(* ---------------------- Limitation of the command signal between +/- SpeedLimit ----------------------------*)
IF fL_CommandSignal > (fI_SpeedLimit) THEN
  fL_CommandSignal :=  fI_SpeedLimit;
ELSIF fL_CommandSignal < (-fI_SpeedLimit) THEN
  fL_CommandSignal := -fI_SpeedLimit;
END_IF;

IF bI_MoveEnable THEN
  IF fI_Microstepping <> 0 THEN
    iO_TargetVelocity := FC_REAL_TO_INT((fI_LimitSpeedFullStep / (fI_LimitSpeedFullStep / fI_Microstepping / 60 * fI_Axis_Scaling) * fL_CommandSignal * fL_PercentageRampUP)); 
    //iO_TargetVelocity := FC_REAL_TO_INT((fI_SpeedScaling / fI_Axis_Scaling * fL_CommandSignal * fL_PercentageRampUP));      (* Send the Target velocity command to module *)
  END_IF;
ELSE
  IF fI_Microstepping <> 0 THEN
    iO_TargetVelocity := FC_REAL_TO_INT((fI_LimitSpeedFullStep / (fI_LimitSpeedFullStep / fI_Microstepping / 60 * fI_Axis_Scaling) * fL_CommandSignal * (1-fL_PercentageRampDN))); 
    //iO_TargetVelocity := FC_REAL_TO_INT((fI_SpeedScaling / fI_Axis_Scaling * fL_CommandSignal * (1-fL_PercentageRampDN)));  (* Send the Target velocity command to module *)
  END_IF;
END_IF;

IF NOT bI_EStop THEN
  iO_TargetVelocity := 0;
END_IF;


(* ---------------------- Encoder Offset Calibration ----------------- *)

IF bI_SetPosition AND NOT bL_memSetPosition AND NOT bI_MoveEnable THEN
  IF fI_Axis_Scaling <> 0 THEN
    fL_OffsetEncoder := FC_REAL_TO_DINT((fI_SetPositionValue * fI_EncoderScaling / fI_Axis_Scaling - DINT_TO_REAL(lI_EncoderValue)));
  END_IF;

  fL_memTargetPosition := fO_ActualPosition;
END_IF;

(* ---------------------- Memory ----------------- *)
bL_memSetPosition := bI_SetPosition;
bL_memMoveEnable  := bI_MoveEnable;
bL_FirstRun       := FALSE;

(********************************* END OF FB *****************************************************)

METHOD PRIVATE Input
VAR_INPUT
END_VAR
(*EL7041 Standard: 20 Singleturn bits and 12 Multiturn bits*)
IF (fI_EncoderScaling <> 0) THEN
	fO_ActualPosition := (DINT_TO_REAL(lI_EncoderValue) + DINT_TO_REAL(fL_OffsetEncoder)) * fI_Axis_Scaling / fI_EncoderScaling;
END_IF;

(*Movement done?*)
IF bI_MoveEnable THEN
	IF ABS(fL_memTargetPosition - fO_ActualPosition) < fI_Tolerance * 0.2 THEN
		bO_MoveOK := TRUE;
	ELSE
		bO_MoveOK := FALSE;
	END_IF;
ELSE
	IF ABS(fL_memTargetPosition - fO_ActualPosition) < fI_Tolerance THEN
		bO_MoveOK := TRUE;
	ELSE
		bO_MoveOK := FALSE;
	END_IF;
END_IF;
END_METHOD

END_FUNCTION_BLOCK

// ---- POUs/Machine/CleaningStation/FB_EL7201_001_AXIS_CTRL.TcPOU
FUNCTION_BLOCK FB_EL7201_001_AXIS_CTRL
(*************************************************************************************************)
(*  FILENAME:    FB_EL7201_001_AXIS_CTRL.EXP                                                     *)
(*  PROJECT:     CALMAR PUPLC                                                                    *)
(*  COPYRIGHT:   All rights reserved (c) Wifag//Polytype, Fribourg/Switzerland (2016)            *)
(*  ENVIRONMENT: TwinCAT PLC                                                                     *)
(*  VERSION:     <version>                                                                       *)
(*************************************************************************************************)
(*  DESCRIPTION:                                                                   <description> *)
(*     This function transfers the movement commands to the motor.                               *)
(*     It also controls the states of the EL7201 for the Cleaning Unit.                          *)
(*                                                                                </description> *)
(*************************************************************************************************)

{library public}
VAR_INPUT
  fI_TargetPosition              : REAL;                         (*Target position*)
  fI_Tolerance                   : REAL := 0.00002;              (*Position tolerance*)
  fI_SpeedLimit                  : REAL;                         (*Speed limit*)
  bI_MoveEnable                  : BOOL;                         (*Enable movement*)
  bI_RegActive                   : BOOL;                         (*Regulation active*)
  bI_FaultReset                  : BOOL;                         (*Fault reset*)
  bI_EStop                       : BOOL;                         (*Emergency stop*)
  bI_SetPosition                 : BOOL;                         (*Set position*)

  wI_StatusWord                  : UINT;                         (*Status word: 6041:0*)
  lI_EncoderValue                : UDINT;                        (*Encoder value*)
  fI_PosControllerGain           : REAL := 1.0;                  (*Position controller gain*)
  fI_EncoderScaling              : REAL := 1048576;              (*Encoder scaling [counts/rev]*)
  fI_Axis_Scaling                : REAL := 0.0002;               (*Axis scaling [m/rev]*)
  fI_SetPositionValue            : REAL := 0.0;                  (*Set position value [m]*)
  fI_SpeedScaling                : REAL := 268435;               (*Speed scaling [counts/rev]*)

  pI_OffsetEncoder               : POINTER TO DINT;              (*Offset to remanent value in encoder*)
END_VAR

VAR_OUTPUT
  wO_ControlWord                 : UINT;                         (*Control word:  6040:0*)
  iO_TargetVelocity              : DINT;                         (*Target velocity:  60FF:0*)
  fO_ActualPosition              : REAL;                         (*Actual position [m]*)
  bO_MoveOk                      : BOOL;                         (*Movement ok*)
  eO_EL7201Status                : EN_EL7201_STATE;              (*EL7201 Status*)
  bO_AxisNotInit                 : BOOL;                         (*Axis not initialized*)
END_VAR

{library private}
VAR
  fL_Delta_P                     : REAL;                         (*Delta position*)
  fL_CommandSignal               : REAL;                         (*Command signal*)

  tL_TimerRampUP                 : TON;                          (*Timer ramp up*)
  fL_PercentageRampUP            : REAL;                         (*Percentage ramp up*)
  tL_TimerRampDN                 : TON;                          (*Timer ramp down*)
  fL_PercentageRampDN            : REAL;                         (*Percentage ramp down*)

  wL_MaskedStatusWord            : WORD;                         (*Masked status word*)
  bL_memMoveEnable               : BOOL;                         (*Memory enable movement*)
  bL_memSetPosition              : BOOL;                         (*Memory set position*)
  fL_memTargetPosition           : REAL := 0.0;                  (*Memory target position*)
  bL_StopRamp                    : BOOL;                         (*Stop ramp*)
  bL_FirstRun                    : BOOL := TRUE;                 (*First run*)

  fL_Divider                     : REAL;                         (*Divider for percent calculation*)
END_VAR

Input();

tL_TimerRampUP.PT :=T#100ms;
tL_TimerRampUP();

tL_TimerRampDN.PT :=T#100ms;
tL_TimerRampDN();

IF bI_MoveEnable=FALSE AND bL_memMoveEnable THEN
	bL_StopRamp := TRUE;
END_IF;

IF bI_MoveEnable AND NOT bL_memMoveEnable THEN
	fL_memTargetPosition := fI_TargetPosition;
	bO_MoveOK := FALSE;
ELSIF bL_FirstRun THEN
	fL_memTargetPosition := fO_ActualPosition;
END_IF;


IF tL_TimerRampDN.Q THEN
	bL_StopRamp:=FALSE;
END_IF;

tL_TimerRampDN.IN := bL_StopRamp;

fL_Divider := TIME_TO_REAL(tL_TimerRampDN.PT);
IF fL_Divider <> 0 THEN
	fL_PercentageRampDN := TIME_TO_REAL(tL_TimerRampDN.ET)/fL_Divider;
END_IF;

tL_TimerRampUP.IN := bI_MoveEnable AND bI_RegActive;

fL_Divider := TIME_TO_REAL(tL_TimerRampUP.PT);
IF fL_Divider <> 0 THEN
	fL_PercentageRampUP := TIME_TO_REAL(tL_TimerRampUP.ET)/fL_Divider;
END_IF;

(* ---------------------- Calculation of the Error Signal between the Target and the Actual Position -----------------*)
fL_Delta_P := fI_TargetPosition - fO_ActualPosition;

(* --------------------------------- Calculation of the Command Signal for the Target Velocity  ---------------------------*)
fL_CommandSignal := fL_Delta_P * fI_PosControllerGain;

(* ----------------------------- Limitation of the Command Signal between +/- SpeedLimit --------------------------------*)
IF fL_CommandSignal > (fI_SpeedLimit) THEN
	fL_CommandSignal:= fI_SpeedLimit;
ELSIF fL_CommandSignal < (-fI_SpeedLimit) THEN
	fL_CommandSignal:=-fI_SpeedLimit;
END_IF;

IF bI_MoveEnable THEN
	IF fI_Axis_Scaling <> 0 THEN
		iO_TargetVelocity:= FC_REAL_TO_DINT((fI_SpeedScaling / fI_Axis_Scaling * fL_CommandSignal * fL_PercentageRampUP));			(* Send the Target velocity command to module *)
	END_IF;
ELSE
	IF fI_Axis_Scaling <> 0 THEN
		iO_TargetVelocity:= FC_REAL_TO_DINT((fI_SpeedScaling / fI_Axis_Scaling * fL_CommandSignal * (1-fL_PercentageRampDN)));	(* Send the Target velocity command to module *)
	END_IF;
END_IF;
(* ---------------------- MDP StateMachine ----------------- *)

wL_MaskedStatusWord := UINT_TO_WORD(wI_StatusWord) AND 16#006F;

IF bI_EStop=FALSE THEN
	iO_TargetVelocity:=0;
	eO_EL7201Status := eEstopped;
	wO_ControlWord := 16#0000;
	wO_ControlWord := 16#0002;
ELSE

	CASE wL_MaskedStatusWord OF
			16#0000, 16#0020:								(* ------------------ State : Not Ready to Switch On : x0xx0000 ---------------------- *)
				eO_EL7201Status := eNotReadyToSwitchON ;

			16#0040, 16#0060:								(* ------------------ State : Switch ON Disable : x1xx0000 ---------------------- *)
				eO_EL7201Status := eSwitchONDisabled ;
				wO_ControlWord := 16#0006;

			16#0021:										(* ------------------ State : Ready To Switch ON : x01x0001---------------------- *)
				eO_EL7201Status := eReadyToSwitchON ;
				IF bI_RegActive=TRUE THEN
					wO_ControlWord := 16#0007;
				ELSE
					wO_ControlWord := 16#0006;
				END_IF;

			16#0023:										(* ---------------- State : Switched ON : x01x0011------------------ *)
				eO_EL7201Status := eSwitchedON ;
				IF bI_MoveEnable=TRUE THEN
					wO_ControlWord := 16#000F;
				END_IF;

				IF bI_RegActive=FALSE THEN
					wO_ControlWord := 16#0006;
				END_IF;

			16#0027:										(* -------------- State : Enabled : x01x0111------------------ *)
				eO_EL7201Status := eEnabled;
				IF (bI_MoveEnable=FALSE AND tL_TimerRampDN.Q) THEN
					wO_ControlWord := 16#0007;
				END_IF;

			16#000F, 16#002F:								(* -------------- State : Fault Reaction Active : x0xx1111----------------- *)
				eO_EL7201Status := eFaultReactionActive ;

			16#0008, 16#0028, 16#0068:								(* --------------- State :  Fault : x0xx1000 ------------------- *)
				eO_EL7201Status := eFault;
				IF bI_FaultReset THEN
					wO_ControlWord := 16#0080;
				ELSE
					wO_ControlWord := 16#0000;
				END_IF;
	END_CASE;
END_IF;

(* ---------------------- Encoder Offset Calibration ----------------- *)

IF bI_SetPosition AND NOT bL_memSetPosition AND NOT bI_MoveEnable THEN
	IF fI_Axis_Scaling <> 0 THEN
		pI_OffsetEncoder^:= FC_REAL_TO_DINT((fI_SetPositionValue * fI_EncoderScaling / fI_Axis_Scaling - UDINT_TO_REAL(lI_EncoderValue)));
	END_IF;

	fL_memTargetPosition := fO_ActualPosition;
END_IF;

IF pI_OffsetEncoder^ = 0 OR pI_OffsetEncoder = 0 THEN
	bO_AxisNotInit := TRUE;
ELSE
	bO_AxisNotInit := FALSE;
END_IF;

(* ---------------------- Memory ----------------- *)
bL_memSetPosition := bI_SetPosition;
bL_memMoveEnable  := bI_MoveEnable;
bL_FirstRun       := FALSE;

(********************************* END OF FB *****************************************************)

ACTION Input:
(*EL7201 Standard: 20 Singleturn bits and 12 Multiturn bits*)
IF fI_EncoderScaling <> 0 AND pI_OffsetEncoder <> 0 THEN
	fO_ActualPosition:=(UDINT_TO_REAL(lI_EncoderValue) + DINT_TO_REAL(pI_OffsetEncoder^)) * fI_Axis_Scaling / fI_EncoderScaling;
END_IF;

(*Movement done?*)
IF ABS(fL_memTargetPosition - fO_ActualPosition) < fI_Tolerance THEN
	bO_MoveOK := TRUE;
ELSE
	bO_MoveOK := FALSE;
END_IF;

(********************************* END OF ACTION *************************************************)
END_ACTION

END_FUNCTION_BLOCK

// ---- POUs/Machine/CleaningStation/FB_EL7201_AXIS_CTRL.TcPOU
FUNCTION_BLOCK FB_EL7201_AXIS_CTRL
(*************************************************************************************************)
(*  FILENAME:    FB_EL7201_AXIS_CTRL.EXP                                                         *)
(*  PROJECT:     CALMAR PUPLC                                                                    *)
(*  COPYRIGHT:   All rights reserved (c) Wifag//Polytype, Fribourg/Switzerland (2016)            *)
(*  ENVIRONMENT: TwinCAT PLC                                                                     *)
(*  VERSION:     <version>                                                                       *)
(*************************************************************************************************)
(*  DESCRIPTION:                                                                   <description> *)
(*     This function transfers the movement commands to the motor.                               *)
(*     It also controls the states of the EL7201 for the Cleaning Unit.                          *)
(*                                                                                </description> *)
(*************************************************************************************************)

{library public}
VAR_INPUT
  fI_TargetPosition              : REAL;                         (*Target position*)
  fI_Tolerance                   : REAL := 0.0001;               (*Position tolerance*)
  fI_SpeedLimit                  : REAL;                         (*Speed limit*)
  bI_MoveEnable                  : BOOL;                         (*Enable movement*)
  bI_RegActive                   : BOOL;                         (*Regulation active*)
  bI_FaultReset                  : BOOL;                         (*Fault reset*)
  bI_MsgReset                    : BOOL;                         (*Message reset*)
  bI_EStop                       : BOOL;                         (*Emergency stop*)
  bI_SetPosition                 : BOOL;                         (*Set position*)

  wI_StatusWord                  : UINT;                         (*Status word: 6041:0*)
  lI_EncoderValue                : DINT;                         (*Encoder value*)
  fI_PosControllerGain           : REAL := 1.0;                  (*Position controller gain*)
  fI_EncoderScaling              : REAL := 1048576;              (*Encoder scaling [counts/rev]*)
  fI_Axis_Scaling                : REAL := 0.0002;               (*Axis scaling [m/rev]*)
  fI_SetPositionValue            : REAL := 0.0;                  (*Set position value [m]*)
  fI_SpeedScaling                : REAL := 268435;               (*Speed scaling [counts/rev]*)

  pI_OffsetEncoder               : POINTER TO DINT;              (*Offset to remanent value in encoder*)

  fI_TolDriveTimeFactor          : REAL := 2.0;                  (*Factor for tolerated drive time*)
END_VAR

VAR_OUTPUT
  wO_ControlWord                 : UINT;                         (*Control word:  6040:0*)
  iO_TargetVelocity              : DINT;                         (*Target velocity:  60FF:0*)
  fO_ActualPosition              : REAL;                         (*Actual position [m]*)
  bO_MoveOk                      : BOOL;                         (*Movement ok*)
  eO_EL7201Status                : EN_EL7201_STATE;              (*EL7201 status*)
  bO_WarnDriveTime               : BOOL;                         (*Error drive time too long*)
END_VAR

{library private}
VAR
  fL_Delta_P                     : REAL;                         (*Delta position*)
  fL_CommandSignal               : REAL;                         (*Command signal*)

  tL_TimerRampUP                 : TON;                          (*Timer ramp up*)
  fL_PercentageRampUP            : REAL;                         (*Percentage ramp up*)
  tL_TimerRampDN                 : TON;                          (*Timer ramp down*)
  fL_PercentageRampDN            : REAL;                         (*Percentage ramp down*)

  wL_MaskedStatusWord            : WORD;                         (*Masked status word*)
  bL_memMoveEnable               : BOOL;                         (*Memory enable movement*)
  bL_memSetPosition              : BOOL;                         (*Memory set position*)
  fL_memTargetPosition           : REAL := 0.0;                  (*Memory target position*)
  bL_StopRamp                    : BOOL;                         (*Stop ramp*)
  bL_FirstRun                    : BOOL := TRUE;                 (*First run*)

  fL_Divider                     : REAL;                         (*Divider for percent calculation*)
  
  fb_RTrigEnable                 : R_TRIG;                       (*RTrig for motor enable*)
  fL_CalcDriveTime               : REAL;                         (*Calculated drive time [s]*)
  fL_RampDriveTime               : REAL := 10;                   (*Ramp time [s]*)
  tL_DriveTime                   : TON;                          (*Timer drive time*)
  iL_SpeedNotSetCounter          : UINT;                         (*Debug: speed limit for calculation not set*)
END_VAR

Input();

tL_TimerRampUP.PT :=T#300ms;
tL_TimerRampUP();

tL_TimerRampDN.PT :=T#300ms;
tL_TimerRampDN();

IF bI_MoveEnable=FALSE AND bL_memMoveEnable=TRUE THEN
	bL_StopRamp := TRUE;
END_IF;

IF bI_MoveEnable=TRUE AND bL_memMoveEnable=FALSE THEN
	fL_memTargetPosition := fI_TargetPosition;
	bO_MoveOK := FALSE;
ELSIF bL_FirstRun THEN
	fL_memTargetPosition := fO_ActualPosition;
END_IF;


IF tL_TimerRampDN.Q THEN
	bL_StopRamp:=FALSE;
END_IF;

tL_TimerRampDN.IN := bL_StopRamp;

fL_Divider := TIME_TO_REAL(tL_TimerRampDN.PT);
IF fL_Divider <> 0 THEN
	fL_PercentageRampDN := TIME_TO_REAL(tL_TimerRampDN.ET)/fL_Divider;
END_IF;

tL_TimerRampUP.IN := bI_MoveEnable AND bI_RegActive;

fL_Divider := TIME_TO_REAL(tL_TimerRampUP.PT);
IF fL_Divider <> 0 THEN
	fL_PercentageRampUP := TIME_TO_REAL(tL_TimerRampUP.ET)/fL_Divider;
END_IF;

(* ---------------------- Calculation of the Error Signal between the Target and the Actual Position -----------------*)
fL_Delta_P := fI_TargetPosition - fO_ActualPosition;

(* --------------------------------- Calculation of the Command Signal for the Target Velocity  ---------------------------*)
fL_CommandSignal := fL_Delta_P * fI_PosControllerGain;

(* ----------------------------- Limitation of the Command Signal between +/- SpeedLimit --------------------------------*)
IF fL_CommandSignal > (fI_SpeedLimit) THEN
	fL_CommandSignal:= fI_SpeedLimit;
ELSIF fL_CommandSignal < (-fI_SpeedLimit) THEN
	fL_CommandSignal:=-fI_SpeedLimit;
END_IF;

IF bI_MoveEnable THEN
	IF fI_Axis_Scaling <> 0 THEN
		iO_TargetVelocity:= FC_REAL_TO_DINT((fI_SpeedScaling / fI_Axis_Scaling * fL_CommandSignal * fL_PercentageRampUP));			(* Send the Target velocity command to module *)
	END_IF;
ELSE
	IF fI_Axis_Scaling <> 0 THEN
		iO_TargetVelocity:= FC_REAL_TO_DINT((fI_SpeedScaling / fI_Axis_Scaling * fL_CommandSignal * (1-fL_PercentageRampDN)));	(* Send the Target velocity command to module *)
	END_IF;
END_IF;
(* ---------------------- MDP StateMachine ----------------- *)

wL_MaskedStatusWord := UINT_TO_WORD(wI_StatusWord) AND 16#006F;

IF bI_EStop=FALSE THEN
	iO_TargetVelocity:=0;
	eO_EL7201Status := eEstopped;
	wO_ControlWord := 16#0000;
	wO_ControlWord := 16#0002;
ELSE

	CASE wL_MaskedStatusWord OF
			16#0000, 16#0020:								(* ------------------ State : Not Ready to Switch On : x0xx0000 ---------------------- *)
				eO_EL7201Status := eNotReadyToSwitchON ;

			16#0040, 16#0060:								(* ------------------ State : Switch ON Disable : x1xx0000 ---------------------- *)
				eO_EL7201Status := eSwitchONDisabled ;
				wO_ControlWord := 16#0006;

			16#0021:										(* ------------------ State : Ready To Switch ON : x01x0001---------------------- *)
				eO_EL7201Status := eReadyToSwitchON ;
				IF bI_RegActive=TRUE THEN
					wO_ControlWord := 16#0007;
				END_IF;

			16#0023:										(* ---------------- State : Switched ON : x01x0011------------------ *)
				eO_EL7201Status := eSwitchedON ;
				IF bI_MoveEnable=TRUE THEN
					wO_ControlWord := 16#000F;
				END_IF;

				IF bI_RegActive=FALSE THEN
					wO_ControlWord := 16#0006;
				END_IF;

			16#0027:										(* -------------- State : Enabled : x01x0111------------------ *)
				eO_EL7201Status := eEnabled;
				IF (bI_MoveEnable=FALSE AND tL_TimerRampDN.Q) THEN
					wO_ControlWord := 16#0007;
				END_IF;

			16#000F, 16#002F:								(* -------------- State : Fault Reaction Active : x0xx1111----------------- *)
				eO_EL7201Status := eFaultReactionActive ;

			16#0008, 16#0028, 16#0068:								(* --------------- State :  Fault : x0xx1000 ------------------- *)
				eO_EL7201Status := eFault;
				IF bI_FaultReset THEN
					wO_ControlWord := 16#0080;
				ELSE
					wO_ControlWord := 16#0000;
				END_IF;
	END_CASE;
END_IF;

(* ---------------------- Encoder Offset Calibration ----------------- *)

IF bI_SetPosition AND NOT bL_memSetPosition AND NOT bI_MoveEnable THEN
	IF fI_Axis_Scaling <> 0 THEN
		pI_OffsetEncoder^ := FC_REAL_TO_DINT((fI_SetPositionValue * fI_EncoderScaling / fI_Axis_Scaling - DINT_TO_REAL(lI_EncoderValue)));
	END_IF;

	fL_memTargetPosition := fO_ActualPosition;
END_IF;

(* ---------------------- Memory ----------------- *)
bL_memSetPosition := bI_SetPosition;
bL_memMoveEnable  := bI_MoveEnable;
bL_FirstRun       := FALSE;

(* ---------------------- Check motor for stiffness or blocking ----------------- *)
fb_RTrigEnable(CLK := bI_MoveEnable);
IF fb_RTrigEnable.Q THEN
  IF (fI_SpeedLimit <> 0) THEN
    fL_CalcDriveTime := ABS(fL_Delta_P / fI_SpeedLimit);
  ELSE
    fL_CalcDriveTime := 250;  (*SpeedLimit not set in time*)
    iL_SpeedNotSetCounter := iL_SpeedNotSetCounter + 1;
  END_IF

  tL_DriveTime(IN := TRUE, PT := REAL_TO_TIME(((fL_CalcDriveTime * fI_TolDriveTimeFactor) + fL_RampDriveTime) * 1000));
END_IF

IF bI_MoveEnable THEN
  tL_DriveTime();
ELSE
  tL_DriveTime(IN := FALSE);
END_IF

IF tL_DriveTime.Q THEN
  bO_WarnDriveTime := TRUE;
END_IF
IF bI_MsgReset THEN
  bO_WarnDriveTime := FALSE;
END_IF;


(********************************* END OF FB *****************************************************)

ACTION Input:
(*EL7201 Standard: 20 Singleturn bits and 12 Multiturn bits*)
IF (fI_EncoderScaling <> 0) AND (pI_OffsetEncoder <> 0) THEN
	fO_ActualPosition := (DINT_TO_REAL(lI_EncoderValue) + DINT_TO_REAL(pI_OffsetEncoder^)) * fI_Axis_Scaling / fI_EncoderScaling;
END_IF;

(*Movement done?*)
IF bI_MoveEnable THEN
	IF ABS(fL_memTargetPosition - fO_ActualPosition) < fI_Tolerance*0.2 THEN
		bO_MoveOK := TRUE;
	ELSE
		bO_MoveOK := FALSE;
	END_IF;
ELSE
	IF ABS(fL_memTargetPosition - fO_ActualPosition) < fI_Tolerance THEN
		bO_MoveOK := TRUE;
	ELSE
		bO_MoveOK := FALSE;
	END_IF;
END_IF;

(********************************* END OF ACTION *************************************************)
END_ACTION

END_FUNCTION_BLOCK

// ---- POUs/Machine/CleaningStation/FB_EL7342_AXIS_CTRL.TcPOU
FUNCTION_BLOCK FB_EL7342_AXIS_CTRL
(*************************************************************************************************)
(*  FILENAME:    FB_EL7342_AXIS_CTRL.EXP                                                         *)
(*  PROJECT:     CALMAR PUPLC                                                                    *)
(*  COPYRIGHT:   All rights reserved (c) Wifag//Polytype, Fribourg/Switzerland (2016)            *)
(*  ENVIRONMENT: TwinCAT PLC                                                                     *)
(*  VERSION:     <version>                                                                       *)
(*************************************************************************************************)
(*  DESCRIPTION:                                                                   <description> *)
(*     This function transfers the movement commands to the motor.                               *)
(*     It also provide a position control for the Cleaning Head.                                 *)
(*                                                                                </description> *)
(*************************************************************************************************)

{library public}
VAR_INPUT
  (*From Motion Controller*)
  bI_MovePos                     : BOOL;                         (*Movement positive direction*)
  bI_MoveNeg                     : BOOL;                         (*Movement negative direction*)
  fI_SpeedLimit                  : REAL;                         (*Speed limit*)
  bI_MoveEnable                  : BOOL;                         (*Enable movement*)
  bI_RegActive                   : BOOL;                         (*Regulation active*)
  bI_FaultReset                  : BOOL;                         (*Reset the errors*)

  (*From Machine*)
  bI_EStop                       : BOOL;                         (*Emergency stop*)
  bI_PositionReset               : BOOL;                         (*Position reset*)

  (*Inputs from Motor*)
  bI_MotorStatus_ReadyToEnable   : BOOL;                         (*Cleaning Head is powered up*)
  bI_MotorStatus_Ready           : BOOL;                         (*Cleaning Head is ready for new command*)
  bI_MotorStatus_Error           : BOOL;                         (*Motor status error*)

  (*Config*)
  fI_Axis_Scaling                : REAL := 0;                    (*Config axis scaling [m/rev]*)
END_VAR

VAR_OUTPUT
  (*To Motor*)
  iO_Velocity                    : INT;                          (*Defines the rotation speed of the motor*)
  bO_Enable                      : BOOL;                         (*Activates the output stage of the module*)
  bO_Reset                       : BOOL;                         (*Feedback reset error*)

  (*To MotionController*)
  eO_EL7342Status                : EN_EL7342_STATE;              (*EL7342 status*)
  fO_CurrentPosition             : REAL;                         (*Curent position*)
END_VAR

{library private}
VAR
  fb_getSysTime                  : GETSYSTEMTIME;                (*Get system time*)
  iL_TimeStamp                   : DINT;                         (*Time stamp*)
  iL_PrevTimeStamp               : DINT;                         (*Previous time stamp*)
  iL_DeltaTime                   : DINT;                         (*Delta time*)
  iL_ElapsedTime                 : DINT;                         (*Elapsed time*)
  fL_CurrentPosition             : REAL;                         (*Current position*)

  fL_GearBoxRatio                : REAL;                         (*Gear box ratio*)
END_VAR

bO_Reset := bI_FaultReset;		(* Reset the errors if the input is active *)

IF NOT bI_EStop THEN
	bO_Enable       := FALSE;
	iO_Velocity     := 0;
	eO_EL7342Status := eEmergencyStopped;

ELSIF bI_MotorStatus_Error THEN							(* If the Motor is faulty*)
	eO_EL7342Status := eFaulty;
	(* ADD ERROR CODE TREATMENT *)

ELSIF bI_MotorStatus_ReadyToEnable THEN			(* When the Output Stage is ready to be Enabled *)
	eO_EL7342Status := eReadyToEnable;

	IF (bI_MotorStatus_Ready OR bI_MotorStatus_ReadyToEnable) AND fI_Axis_Scaling <> 0 THEN
		iO_Velocity := FC_REAL_TO_INT(MIN(fI_SpeedLimit * 1000 * (32767 / fI_Axis_Scaling), 32767));	(* Speed Setup for the mouvement *)

		IF bI_MovePos AND NOT bI_MoveNeg THEN
			eO_EL7342Status := eStarted;
			iO_Velocity     := -iO_Velocity;
		ELSIF NOT bI_MovePos AND bI_MoveNeg THEN
			eO_EL7342Status := eStarted;
			iO_Velocity     := iO_Velocity;
		ELSE
			eO_EL7342Status := eReady;
			iO_Velocity     := 0;
		END_IF;

		bO_Enable := bI_MoveEnable;				(* The mouvement will be executed according to the FB_CH_MOTION_CTRL Command*)
	END_IF;

	IF bI_MoveEnable AND bI_MotorStatus_Ready THEN
		fb_getSysTime();
		iL_TimeStamp := UDINT_TO_DINT(fb_getSysTime.timeLoDW);

		IF iL_PrevTimeStamp <> 0THEN
			iL_DeltaTime := iL_TimeStamp - iL_PrevTimeStamp; (* Give the delta time between two cycles in nanoseconds *)
		END_IF;

		IF bI_MovePos THEN
		(*	fL_CurrentPosition := fL_CurrentPosition + (iL_DeltaTime) * ((fI_SpeedLimit*(fI_Axis_Scaling/32767))/10000000);*)
			fL_CurrentPosition := fL_CurrentPosition + DINT_TO_REAL(iL_DeltaTime) / 10_000_000 * fI_SpeedLimit;
		ELSIF bI_MoveNeg THEN
(*			fL_CurrentPosition := fL_CurrentPosition - (iL_DeltaTime) * ((fI_SpeedLimit*(fI_Axis_Scaling/32767))/10000000);*)
			fL_CurrentPosition := fL_CurrentPosition - DINT_TO_REAL(iL_DeltaTime) / 10_000_000 * fI_SpeedLimit;
		END_IF;
		iL_PrevTimeStamp := iL_TimeStamp;
	ELSE
		iL_PrevTimeStamp := 0;
	END_IF;

	IF bI_PositionReset THEN
		fL_CurrentPosition := 0;
	END_IF;
END_IF;
fO_CurrentPosition := fL_CurrentPosition;

(********************************* END OF FB *****************************************************)

END_FUNCTION_BLOCK

// ---- POUs/Machine/CleaningStation/FB_MachineState.TcPOU
FUNCTION_BLOCK FB_MachineState IMPLEMENTS I_MachineStateBase
(*************************************************************************************************)
(*  FILENAME:    FB_MachineState                                                                 *)
(*  PROJECT:     CALMAR PUPLC                                                                    *)
(*  COPYRIGHT:   All rights reserved (c) Polytype AG, Fribourg/Switzerland (2020)                *)
(*  ENVIRONMENT: TwinCAT PLC                                                                     *)
(*  VERSION:     <version>                                                                       *)
(*************************************************************************************************)
(*  DESCRIPTION:                                                                   <description> *)
(*    add description                                                                            *)
(*                                                                                </description> *)
(*************************************************************************************************)

VAR_INPUT
  bI_SafetyOk                     : BOOL;  (*Safety ok for movement*)
  bI_MachineReady                 : BOOL;  (*Machine ready*)
END_VAR

PROPERTY pMachineReady : BOOL
GET
pMachineReady := bI_MachineReady;
END_GET
END_PROPERTY

PROPERTY pSafetyOk : BOOL
GET
pSafetyOk := bI_SafetyOk;
END_GET
END_PROPERTY

END_FUNCTION_BLOCK

// ---- POUs/Machine/CleaningStation/FB_MOTOR_SWITCH.TcPOU
FUNCTION_BLOCK FB_MOTOR_SWITCH
(*************************************************************************************************)
(*  FILENAME:    FB_MOTOR_SWITCH.EXP                                                             *)
(*  PROJECT:     CALMAR PUPLC                                                                    *)
(*  COPYRIGHT:   All rights reserved (c) Wifag//Polytype, Fribourg/Switzerland (2016)            *)
(*  ENVIRONMENT: TwinCAT PLC                                                                     *)
(*  VERSION:     <version>                                                                       *)
(*************************************************************************************************)
(*  DESCRIPTION:                                                                   <description> *)
(*     Detect change in command, commands from B are only accepted when A is false.              *)
(*                                                                                </description> *)
(*************************************************************************************************)

{library public}
VAR_INPUT
  bI_A                           : BOOL;                         (*Input A, priority input*)
  bI_B                           : BOOL;                         (*Input B*)
  lC_Delay                       : INT := 100;                   (*Delay for switching*)
END_VAR

VAR_OUTPUT
  bO_QA                          : BOOL;                         (*Output A*)
  bO_QB                          : BOOL;                         (*Output B*)
END_VAR

{library private}
VAR
  fb_SwitchTimer                 : TP;                           (*Switching timer*)
  bL_Areg                        : BOOL;                         (*Memory A*)
  bL_Breg                        : BOOL;                         (*Memory B*)
END_VAR

fb_SwitchTimer.PT := INT_TO_TIME(lC_Delay);

(*Detect change in Command, commands from B are only accepted when A is false*)
fb_SwitchTimer.IN:=	(bI_A XOR bL_Areg) OR ((bI_B XOR bL_Breg) AND NOT bI_A);
fb_SwitchTimer();

(*Switch logic, A has priority*)

IF bI_A AND NOT fb_SwitchTimer.Q THEN	(*Enable A*)
	bO_QA := TRUE;
	bO_QB := FALSE;
ELSE
	bO_QA := FALSE;	(*Disable A*)

	IF bI_B AND NOT fb_SwitchTimer.Q THEN	(*Enable B*)
		bO_QB := TRUE;
	ELSE
		bO_QB := FALSE;	(*Disable B*)
	END_IF;

END_IF;

(*Register*)
bL_Areg := bI_A;
bL_Breg := bI_B;

(********************************* END OF FB *****************************************************)

END_FUNCTION_BLOCK

// ---- POUs/Machine/CleaningStation/FB_PU_MOTION_CTRL.TcPOU
FUNCTION_BLOCK FB_PU_MOTION_CTRL
(*************************************************************************************************)
(*  FILENAME:     FB_PU_MOTION_CTRL.EXP                                                          *)
(*  PROJECT:      Steinemann                                                                     *)
(*  COPYRIGHT:    Wifag//Polytype Fribourg                                                       *)
(*  ENVIRONMENT:  TwinCAT PLC / CoDeSys                                                          *)
(*  VERSION:      1.0                                                                            *)
(*  DESCRIPTION:                                                                                 *)
(*    This Function is to control the mouvements of the Printer Unit                             *)
(*    on the Z Axis. It will control the operation type and the service                          *)
(*    mode to send motion commands to the axis                                                   *)
(*  AUTHOR:       M: BOYRAZ, GoConcept                                                           *)
(*************************************************************************************************)
(*  MODIFICATIONS:                                                                               *)
(*************************************************************************************************)
(*  Date        Author   Comments                                                                *)
(*  21.07.2014  HOA      Added using of fI_SheetThickness for print position                     *)
(*************************************************************************************************)

VAR_INPUT
(*Commands from Cleaning Process Controller*)
	sI_CleanDevCmd             : ST_CLEANING_DEV_CMD;	(*Initialize operation*)

(*Settings*)
	sI_SpeedDef_Z              : ST_SPEEDS;
	fI_CurrentPosition         : REAL;					(*Current axis position*)
	fI_WaitingPosition         : REAL := 0.01;	(*Waiting position (Production Mode)*)
	fI_PrintPosition           : REAL := 0.001;	(*Print position (Production Mode)*)
	fI_SheetThickness          : REAL := 0.000;	(*Sheet thickness (Production Mode)*)
	fI_ServicePosition         : REAL := 0.4;		(*Service position (Service Mode)*)
	fI_CleanPosition1          : REAL := 0.325;	(*Cleaning station moving position (Service Mode)*)
	fI_CleanPosition2          : REAL := 0.315;	(*Cleaning position (Service Mode)*)
	fI_PositionTolerance       : REAL := 0.0001;(*Service position (Service Mode)*)

(*User Commands*)
	sI_ManualCommands          : ST_MANUAL_CMD;
	bI_AckFault                : BOOL;	(* Acknowledge errors*)
	bI_Enable                  : BOOL;	(* Enable PrintUnit axis*)

(*Machine Flags*)
	bI_DeviceOnline            : BOOL;	(*Check link to device*)
	bI_LimitSW_UP              : BOOL;	(* Axis upper limit switch*)
	bI_LimitSW_DOWN            : BOOL;	(* Axis lower limit switch*)
	bI_SystemReady             : BOOL;	(*General ready flag*)
	bI_MachineReady            : BOOL;	(*Machine ready = go to print if not in service*)
	bI_MovementAllowed         : BOOL;	(*No collision danger*)
	bI_SafetyOk                : BOOL;	(*Safety ok for movement*)
	eI_ELmodule_State          : EN_EL7201_STATE;	(*Feedback from Axis*)
	bI_Chopper_Error           : BOOL := FALSE;
	bI_Chopper_Overvoltage     : BOOL := FALSE;
	bI_Chopper_Undervoltage    : BOOL := FALSE;
	bI_MoveDone                : BOOL;
	bI_AxisNotInit             : BOOL;
	bI_EmergencyMoveUp         : BOOL;

	pC_MsgInterface            : POINTER TO ST_ADS_MSG_IF;
	iC_BlockId                 : INT;
END_VAR

VAR_OUTPUT
	sO_PrintUnit_Mvt_Status    : ST_PU_STATUS;
	sO_CleanDevStatus          : ST_CLEANING_DEV_STATUS;	(*Initialize operation*)

	fO_TargetPosition          : REAL;	(*Target position for axis*)
	fO_SpeedLimit              : REAL;	(*Speed limit for axis*)
	bO_MoveEnable              : BOOL;	(*Move enable for axis*)
	bO_RegActive               : BOOL;	(*Close control loop for axis*)
	bO_FaultReset              : BOOL;	(*Fault reset for axis*)
END_VAR

VAR
	bL_SafeRunningCondition    : BOOL;
	bL_SafeMoveDown            : BOOL;
	bL_SafeMoveUp              : BOOL;

	bL_AxisReady               : BOOL;	(*Axis has no pending operation*)
	bL_PrintReady              : BOOL;	(*Axis is ready to print*)

	wL_ErrorCode               : WORD;

	fL_PrintPosition           : REAL;	(*Print position (Production Mode)*)

	bL_InPosition_C1           : BOOL;
	bL_InPosition_C2           : BOOL;
	bL_InPosition_Waiting      : BOOL;
	bL_InPosition_Printing     : BOOL;
	bL_InPosition_Service      : BOOL;
	bL_MotionActive            : BOOL;
	bL_SafeMoveRequired        : BOOL := TRUE;
	bL_MoveStarted             : BOOL := FALSE;
	bL_MoveStartRequested      : BOOL := FALSE;
	bL_MoveDone                : BOOL := FALSE;

	tL_TimerSurv               : TON;			(* Timer for Motorization check *)

	(*Memory registers*)
	bL_mem_MotionActive        : BOOL;
	bL_memAckFault             : BOOL;
	fL_memZ_Position           : REAL;
	bL_mem_MoveEnable          : BOOL;
	bL_memLimitSW_UP           : BOOL;
	bL_memLimitSW_DOWN         : BOOL;
	bL_Cdtion_LimitSW_UP       : BOOL;
	bL_memCdtion_LimitSW_UP    : BOOL;
	bL_Cdtion_LimitSW_DOWN     : BOOL;
	bL_memCdtion_LimitSW_DOWN  : BOOL;
	bL_FirstRun                : BOOL := TRUE;

	(*Message Queue*)
 	fB_MsgQueue                : FB_MSG_QUEUE;
	fB_MsgHandler              : FB_MSG_HANDLER;
	sL_MsgConfig               : ST_MSG_CONFIG;
	fB_Msg                     : ARRAY [1..iC_NUM_MSG] OF FB_MESSAGE;
END_VAR

VAR CONSTANT
	iC_NUM_MSG                 : INT := 4;
END_VAR

tL_TimerSurv.PT := T#3s;
tL_TimerSurv();

fL_PrintPosition := fI_PrintPosition + fI_SheetThickness;



(*----------------------------------------------------------------------------------------------------------------------------------------------- *)
(*Position detection*)
(*----------------------------------------------------------------------------------------------------------------------------------------------- *)

IF     (fI_CurrentPosition >= fI_WaitingPosition - fI_PositionTolerance)
   AND (fI_CurrentPosition <= fI_WaitingPosition + fI_PositionTolerance)
THEN
	bL_InPosition_C1        := FALSE;
	bL_InPosition_C2        := FALSE;
	bL_InPosition_Waiting   := TRUE;
	bL_InPosition_Printing  := FALSE;
	bL_InPosition_Service   := FALSE;
ELSIF  (fI_CurrentPosition >= fL_PrintPosition - fI_PositionTolerance)
   AND (fI_CurrentPosition <= fL_PrintPosition + fI_PositionTolerance)
THEN
	bL_InPosition_C1        := FALSE;
	bL_InPosition_C2        := FALSE;
	bL_InPosition_Waiting   := FALSE;
	bL_InPosition_Printing  := TRUE;
	bL_InPosition_Service   := FALSE;
ELSIF  (fI_CurrentPosition >= fI_ServicePosition - fI_PositionTolerance)
   AND (fI_CurrentPosition <= fI_ServicePosition + fI_PositionTolerance)
THEN
	bL_InPosition_C1        := FALSE;
	bL_InPosition_C2        := FALSE;
	bL_InPosition_Waiting   := FALSE;
	bL_InPosition_Printing  := FALSE;
	bL_InPosition_Service   := TRUE;
ELSIF  (fI_CurrentPosition >= fI_CleanPosition1 - fI_PositionTolerance)
   AND (fI_CurrentPosition <= fI_CleanPosition1 + fI_PositionTolerance)
THEN
	bL_InPosition_C1        := TRUE;
	bL_InPosition_C2        := FALSE;
	bL_InPosition_Waiting   := FALSE;
	bL_InPosition_Printing  := FALSE;
	bL_InPosition_Service   := FALSE;
ELSIF  (fI_CurrentPosition >= fI_CleanPosition2 - fI_PositionTolerance)
   AND (fI_CurrentPosition <= fI_CleanPosition2 + fI_PositionTolerance)
THEN
	bL_InPosition_C1        := FALSE;
	bL_InPosition_C2        := TRUE;
	bL_InPosition_Waiting   := FALSE;
	bL_InPosition_Printing  := FALSE;
	bL_InPosition_Service   := FALSE;
ELSE
	bL_InPosition_C1        := FALSE;
	bL_InPosition_C2        := FALSE;
	bL_InPosition_Waiting   := FALSE;
	bL_InPosition_Printing  := FALSE;
	bL_InPosition_Service   := FALSE;
END_IF;

(*If the axis has been moved above the waiting position, a deblocking move is required before entering print state*)
IF fI_CurrentPosition > fI_WaitingPosition+fI_PositionTolerance THEN
	bL_SafeMoveRequired := TRUE;		(*This flag is cleared in production mode*)
END_IF;

(*----------------------------------------------------------------------------------------------------------------------------------------------- *)
(*----------------------------------- Safe Running Conditions  For Printing Unit  -------------------------------------------- *)
(*----------------------------------------------------------------------------------------------------------------------------------------------- *)
IF bI_Enable AND bI_SystemReady AND bI_DeviceOnline AND bI_SafetyOk AND (wL_ErrorCode = 0 OR wL_ErrorCode.5 OR wL_ErrorCode.6)THEN	(*Dont check limit switch here*)
	bL_SafeRunningCondition := TRUE;
ELSE
	bL_SafeRunningCondition := FALSE;
END_IF;
bL_SafeMoveDown := bL_SafeRunningCondition AND NOT bI_LimitSW_Down AND bI_MovementAllowed;
bL_SafeMoveUp 	:= bL_SafeRunningCondition AND NOT bI_LimitSW_Up;

(*----------------------------------------------------------------------------------------------------------------------------------------------- *)
(* Printer Unit Mouvement Control 																																																								*)
(*----------------------------------------------------------------------------------------------------------------------------------------------- *)
IF sI_CleanDevCmd.bService THEN
	ServiceMode();
ELSE		(* IN PRODUCTION *)
	ProductionMode();
END_IF;


(*----------------------------------------------------------------------------------------------------------------------- *)
(*----------------------------------- Output Structure Data Update  --------------------------------------- *)
(*----------------------------------------------------------------------------------------------------------------------- *)
sO_CleanDevStatus.bBusy     := NOT(bL_AxisReady);
sO_CleanDevStatus.bReady    := bL_AxisReady;
sO_CleanDevStatus.bRefKnown := NOT bI_AxisNotInit;

IF wL_ErrorCode = 0 THEN
	sO_CleanDevStatus.bError := FALSE;
ELSE
	sO_CleanDevStatus.bError := TRUE;
END_IF;

sO_PrintUnit_Mvt_Status.bO_Active              := bI_Enable;
sO_PrintUnit_Mvt_Status.bO_Busy                := bO_MoveEnable;
sO_PrintUnit_Mvt_Status.bO_Ready               := bL_AxisReady;
sO_PrintUnit_Mvt_Status.fO_Position            := fI_CurrentPosition;
sO_PrintUnit_Mvt_Status.bO_InPosition_C1       := bL_InPosition_C1;
sO_PrintUnit_Mvt_Status.bO_InPosition_C2       := bL_InPosition_C2;
sO_PrintUnit_Mvt_Status.bO_InPosition_Printing := bL_InPosition_Printing;
sO_PrintUnit_Mvt_Status.bO_InPosition_Service  := bL_InPosition_Service;
sO_PrintUnit_Mvt_Status.bO_InPosition_Waiting  := bL_InPosition_Waiting;
sO_PrintUnit_Mvt_Status.wO_FaultCode           := wL_ErrorCode;

bO_FaultReset := bI_AckFault (*OR fb_MsgQueue.bO_ReceiptMessage*) OR sI_CleanDevCmd.bAckError;

IF wL_ErrorCode = 0 THEN
	sO_PrintUnit_Mvt_Status.bO_Error := FALSE;
ELSE
	sO_PrintUnit_Mvt_Status.bO_Error := TRUE;
END_IF;

bO_RegActive := bI_Enable AND  bL_SafeRunningCondition;

IF fI_CurrentPosition < fO_TargetPosition THEN			(*  is UP Mouvement *)
	bO_MoveEnable := bL_MotionActive AND bL_SafeMoveUp;
ELSE											(*  is DOWN Mouvement *)
	bO_MoveEnable := bL_MotionActive AND bL_SafeMoveDown;
END_IF;

IF bL_MotionActive AND NOT bL_mem_MotionActive THEN
	bL_MoveStartRequested := TRUE;
	bL_MoveStarted        := FALSE;
	bL_MoveDone           := FALSE;
END_IF;

IF bO_MoveEnable AND NOT bL_mem_MoveEnable AND bL_MoveStartRequested THEN
	bL_MoveStarted := TRUE;
	bL_MoveDone    := FALSE;
ELSIF bL_MoveStarted THEN
	IF bI_MoveDone OR sI_CleanDevCmd.bAbort THEN
		bL_MoveDone           := TRUE;
		bL_MoveStarted        := FALSE;
		bL_MoveStartRequested := FALSE;
	END_IF;
END_IF;

(*----------------------------------------------------------------------------------------------------------------------- *)
(*--------------------------------- Fault Diagnosis and Management  ---------------------------------- *)
(*----------------------------------------------------------------------------------------------------------------------- *)
(*Messaging*)
fB_MsgHandler();

IF eI_ELmodule_State = eFault THEN
  fB_Msg[1].bI_Status := TRUE;
ELSE
  fB_Msg[1].bI_Status := FALSE;
END_IF;
fB_Msg[1]();

fB_Msg[2](bI_Status := bI_Chopper_Error);
fB_Msg[3](bI_Status := bI_Chopper_Overvoltage);
fB_Msg[4](bI_Status := bI_Chopper_Undervoltage);


fB_MsgQueue();



IF (bI_AckFault OR sI_CleanDevCmd.bAckError) AND NOT bL_memAckFault THEN
	tL_TimerSurv.IN := FALSE;
END_IF;

IF bI_AckFault (*OR fb_MsgQueue.bO_ReceiptMessage*) OR sI_CleanDevCmd.bAckError THEN
	wL_ErrorCode := 0;
END_IF;


IF bO_MoveEnable AND NOT bL_mem_MoveEnable THEN
	tL_TimerSurv.IN  := TRUE;
	fL_memZ_Position := fI_CurrentPosition;
END_IF;


IF tL_TimerSurv.Q THEN
	IF NOT bO_MoveEnable THEN			(* If the mouvement is stopped, reset the startup monitoring timer *)
		tL_TimerSurv.IN := FALSE;
	END_IF;
	IF bO_MoveEnable AND (fL_memZ_Position <> fI_CurrentPosition) THEN
		tL_TimerSurv.IN := FALSE;
	END_IF;
END_IF;

IF bI_AxisNotInit THEN
	wL_ErrorCode.1  := TRUE;						(* Axis has lost its value *)
END_IF;
(*
IF bL_MotionActive AND tL_TimerSurv.Q AND (fL_memZ_Position = fI_CurrentPosition) THEN			(* Motorization Fault, Command is active but position is not changing *)
	wL_ErrorCode.2  := TRUE;
END_IF;
*)
IF (sI_SpeedDef_Z.fP_PlaceSpeed = 0) OR (sI_SpeedDef_Z.fP_WorkSpeed = 0) OR (sI_SpeedDef_Z.fP_ServiceSpeed = 0) THEN	(* Speed Configuration not done *)
	wL_Errorcode.3  := TRUE;
END_IF;

IF (fL_PrintPosition = 0) OR (fI_ServicePosition = 0) OR (fI_CleanPosition1 = 0) OR (fI_CleanPosition2 = 0)THEN		(* Position Configuration not done *)
	wL_ErrorCode.4  := TRUE;
END_IF;

IF bI_LimitSW_UP AND NOT bL_memLimitSW_UP THEN
	wL_ErrorCode.5  := TRUE;						(* Safety Fault : Limit Switch UP activated *)
END_IF;

IF bI_LimitSW_DOWN AND NOT bL_memLimitSW_DOWN THEN
	wL_ErrorCode.6  := TRUE;						(* Safety Fault : Limit Switch DOWN activated *)
END_IF;

IF bI_LimitSW_UP AND bI_LimitSW_DOWN THEN
	wL_ErrorCode.7  := TRUE;						(* Safety Fault : Sensor discordance, both Limit Switch UP and DOWN are activated *)
END_IF;

bL_Cdtion_LimitSW_UP := fI_CurrentPosition > (fI_ServicePosition + 0.020);	(*@@@@@@@CONSTANT VALUE*)
IF bL_Cdtion_LimitSW_UP AND NOT bL_memCdtion_LimitSW_UP THEN
	wL_ErrorCode.8  := TRUE;						(* Safety Fault : Limit Switch UP expected *)
END_IF;

bL_Cdtion_LimitSW_DOWN := fI_CurrentPosition < (fL_PrintPosition - 0.020); (*@@@@@@@CONSTANT VALUE*)
IF bL_Cdtion_LimitSW_DOWN AND NOT bL_memCdtion_LimitSW_DOWN THEN
	wL_ErrorCode.9  := TRUE;						(* Safety Fault : Limit Switch DOWN expected *)
END_IF;

IF (eI_ELmodule_State = eFault) OR NOT bI_DeviceOnline THEN
	wL_ErrorCode.10 := TRUE;						(* EL7201 module fault *)
END_IF;
(*
IF NOT bI_SafetyCoversON AND bL_mem_SafetyCoversON  THEN
	wL_ErrorCode.14 := TRUE;						(* Safety Fault *)
END_IF;
*)
(*
IF eI_ELmodule_State = eEstopped THEN
	wL_ErrorCode.15 := TRUE;						(* EL7201 Emergency Stop*)
END_IF;
*)

bL_mem_MotionActive       := bL_MotionActive;
bL_mem_MoveEnable         := bO_MoveEnable;
bL_memAckFault            := bI_AckFault (*OR fb_MsgQueue.bO_ReceiptMessage*) OR sI_CleanDevCmd.bAckError;
bL_memLimitSW_UP          := bI_LimitSW_UP;
bL_memLimitSW_DOWN        := bI_LimitSW_DOWN;
bL_memCdtion_LimitSW_UP   := bL_Cdtion_LimitSW_UP;
bL_memCdtion_LimitSW_DOWN := bL_Cdtion_LimitSW_DOWN;

ACTION Init:
	(*Messages*)
	sL_MsgConfig.bI_Enable       := TRUE;
	sL_MsgConfig.pI_FbMsgHandler := ADR(fB_MsgHandler);
	fB_MsgHandler.pI_MsgQueue    := ADR(fB_MsgQueue);
	fB_MsgQueue.pI_MsgInterface  := pC_MsgInterface;
	fB_MsgQueue.cI_MaxElement    := 5;

	fB_Msg[1].iI_MsgLocation     := iC_BlockId;
	fB_Msg[1].pI_MsgConfig       := ADR(sL_MsgConfig);
	fB_Msg[1].iI_MsgNumber       := eCMa_AxisErrorZ;

	fB_Msg[2].iI_MsgLocation     := iC_BlockId;
	fB_Msg[2].pI_MsgConfig       := ADR(sL_MsgConfig);
	fB_Msg[2].iI_MsgNumber       := eCMa_DC_LINK_ERROR;

	fB_Msg[3].iI_MsgLocation     := iC_BlockId;
	fB_Msg[3].pI_MsgConfig       := ADR(sL_MsgConfig);
	fB_Msg[3].iI_MsgNumber       := eCMa_DC_LINK_OVERVOLTAGE;

	fB_Msg[4].iI_MsgLocation     := iC_BlockId;
	fB_Msg[4].pI_MsgConfig       := ADR(sL_MsgConfig);
	fB_Msg[4].iI_MsgNumber       := eCMa_DC_LINK_UNDERVOLTAGE;
END_ACTION

ACTION ProductionMode:
bL_SafeMoveRequired := FALSE;

IF (fI_CurrentPosition >= fI_WaitingPosition) THEN
	fO_SpeedLimit := sI_SpeedDef_Z.fP_PlaceSpeed;
ELSE
	fO_SpeedLimit := sI_SpeedDef_Z.fP_WorkSpeed;
END_IF;

IF bL_SafeRunningCondition THEN		(* If the Cleaning unit is out of the collision area*)
	IF bI_MachineReady THEN	(*Move to print position*)
		IF    (NOT bL_InPosition_Printing AND NOT bI_EmergencyMoveUp)
       OR (NOT bL_InPosition_Waiting  AND     bI_EmergencyMoveUp)
		THEN
			IF bI_EmergencyMoveUp THEN
				fO_TargetPosition := fI_WaitingPosition;			(* move to WaitingPosition*)
			ELSE
				fO_TargetPosition := fL_PrintPosition;				(* move to PrintPosition*)
			END_IF;
			bL_MotionActive   := TRUE;
			bL_PrintReady     := FALSE;
			bL_AxisReady      := FALSE;
		ELSE
			bL_MotionActive   := FALSE;											(* stop when the position is reached*)
			bL_PrintReady     := TRUE;
			bL_AxisReady      := TRUE;
		END_IF;
	ELSE
		bL_MotionActive := FALSE;
	END_IF;
ELSE
	bL_MotionActive := FALSE;
END_IF;
END_ACTION

ACTION ServiceMode:
(*Default speed*)
IF (fI_CurrentPosition >= fI_WaitingPosition) THEN
	fO_SpeedLimit := sI_SpeedDef_Z.fP_ServiceSpeed;
ELSE
	fO_SpeedLimit := sI_SpeedDef_Z.fP_WorkSpeed;
END_IF;

(*Mode selection*)
IF sI_CleanDevCmd.bAuto THEN	(*Control by cleaning process*)
	CASE 	sI_CleanDevCmd.eOperation OF
		eNOP:	(*No operation active*)
			bL_MotionActive := FALSE;
			bL_AxisReady    := TRUE;

		eOPENDSERVICE: (*End service mode ---------------------------*)
			IF sI_CleanDevCmd.bInit THEN
				IF bL_SafeMoveRequired OR NOT bI_MovementAllowed THEN
					fO_TargetPosition := fI_CleanPosition1;
				ELSE
					fO_TargetPosition := fI_WaitingPosition;
				END_IF;
				bL_MotionActive := TRUE;
				bL_AxisReady    := FALSE;

			ELSIF sI_CleanDevCmd.bPrep THEN
				bL_MotionActive := FALSE;
				bL_AxisReady    := TRUE;

			ELSIF sI_CleanDevCmd.bStart THEN
				bL_MotionActive := FALSE;
				bL_AxisReady    := TRUE;

			ELSIF sI_CleanDevCmd.bStop THEN
				bL_MotionActive := FALSE;
				bL_AxisReady    := TRUE;

			ELSE	(*Command removed, wait until axis finished movement*)
				IF NOT bL_MoveDone THEN
					bL_MotionActive := TRUE;
					bL_AxisReady    := FALSE;
				ELSE
					bL_MotionActive := FALSE;
					bL_AxisReady    := TRUE;
				END_IF;
			END_IF;

		eOPPREPSERVICE, eOPSTARTUP: (*Start service mode ---------------------------*)
			IF sI_CleanDevCmd.bInit THEN
				IF bL_SafeMoveRequired OR sI_CleanDevCmd.eOperation = eOPSTARTUP THEN
					fO_TargetPosition := fI_CleanPosition1;
				ELSE
					fO_TargetPosition := fI_WaitingPosition;
				END_IF;
				bL_MotionActive := TRUE;
				bL_AxisReady    := FALSE;

			ELSIF sI_CleanDevCmd.bPrep THEN
				bL_MotionActive := FALSE;
				bL_AxisReady    := TRUE;

			ELSIF sI_CleanDevCmd.bStart THEN
				bL_MotionActive := FALSE;
				bL_AxisReady    := TRUE;

			ELSIF sI_CleanDevCmd.bStop THEN
				bL_MotionActive := FALSE;
				bL_AxisReady    := TRUE;

			ELSE	(*Command removed, wait until axis finished movement*)
				IF NOT bL_MoveDone THEN
					bL_MotionActive := TRUE;
					bL_AxisReady    := FALSE;
				ELSE
					bL_MotionActive := FALSE;
					bL_AxisReady    := TRUE;
				END_IF;
			END_IF;

		eOPCLEAN:	(*Cleaning Mode -------------------------------------*)
			IF sI_CleanDevCmd.bInit THEN
				fO_TargetPosition := fI_CleanPosition1;
				bL_MotionActive   := TRUE;
				bL_AxisReady      := FALSE;

			ELSIF sI_CleanDevCmd.bPrep THEN
				fO_TargetPosition := fI_CleanPosition2;
				bL_MotionActive   := TRUE;
				bL_AxisReady      := FALSE;

			ELSIF sI_CleanDevCmd.bStart THEN
				bL_MotionActive   := FALSE;
				bL_AxisReady      := TRUE;

			ELSIF sI_CleanDevCmd.bStop THEN
				fO_TargetPosition := fI_CleanPosition1;
				bL_MotionActive   := TRUE;

			ELSE	(*Command removed, wait until axis finished movement*)
				IF NOT bL_MoveDone THEN
					bL_MotionActive := TRUE;
					bL_AxisReady    := FALSE;
				ELSE
					bL_MotionActive := FALSE;
					bL_AxisReady    := TRUE;
				END_IF;
			END_IF;

		eOPPURGE:	(*Purge Mode -------------------------------------*)
			IF sI_CleanDevCmd.bInit THEN
				fO_TargetPosition := fI_CleanPosition1;
				bL_MotionActive   := TRUE;
				bL_AxisReady      := FALSE;

			ELSIF sI_CleanDevCmd.bPrep THEN
				fO_TargetPosition := fI_CleanPosition2;
				bL_MotionActive   := TRUE;
				bL_AxisReady      := FALSE;

			ELSIF sI_CleanDevCmd.bStart THEN
				bL_MotionActive   := FALSE;
				bL_AxisReady      := TRUE;

			ELSIF sI_CleanDevCmd.bStop THEN
				fO_TargetPosition := fI_CleanPosition1;
				bL_MotionActive   := TRUE;

			ELSE	(*Command removed, wait until axis finished movement*)
				IF NOT bL_MoveDone THEN
					bL_MotionActive := TRUE;
					bL_AxisReady    := FALSE;
				ELSE
					bL_MotionActive := FALSE;
					bL_AxisReady    := TRUE;
				END_IF;
			END_IF;

		eOPCAPENTER:	(*Enter Capping Mode -------------------------------------*)
			IF sI_CleanDevCmd.bInit THEN
				fO_TargetPosition := fI_CleanPosition1;
				bL_MotionActive   := TRUE;
				bL_AxisReady      := FALSE;

			ELSIF sI_CleanDevCmd.bPrep THEN
				fO_TargetPosition := fI_CleanPosition2;
				bL_MotionActive   := TRUE;
				bL_AxisReady      := FALSE;

			ELSIF sI_CleanDevCmd.bStart THEN
				bL_MotionActive   := FALSE;
				bL_AxisReady      := TRUE;

			ELSIF sI_CleanDevCmd.bStop THEN
				bL_MotionActive   := FALSE;
				bL_AxisReady      := TRUE;

			ELSE	(*Command removed, wait until axis finished movement*)
				IF NOT bL_MoveDone THEN
					bL_MotionActive := TRUE;
					bL_AxisReady    := FALSE;
				ELSE
					bL_MotionActive := FALSE;
					bL_AxisReady    := TRUE;
				END_IF;
			END_IF;

		eOPCAPEXIT:	(*Exit Capping Mode -------------------------------------*)
			IF sI_CleanDevCmd.bInit THEN
				fO_TargetPosition := fI_CleanPosition1;
				bL_MotionActive   := TRUE;
				bL_AxisReady      := FALSE;

			ELSIF sI_CleanDevCmd.bPrep THEN
				bL_MotionActive   := FALSE;
				bL_AxisReady      := TRUE;

			ELSIF sI_CleanDevCmd.bStart THEN
				bL_MotionActive   := FALSE;
				bL_AxisReady      := TRUE;

			ELSIF sI_CleanDevCmd.bStop THEN
				bL_MotionActive   := FALSE;
				bL_AxisReady      := TRUE;

			ELSE	(*Command removed, wait until axis finished movement*)
				IF NOT bL_MoveDone THEN
					bL_MotionActive := TRUE;
					bL_AxisReady    := FALSE;
				ELSE
					bL_MotionActive := FALSE;
					bL_AxisReady    := TRUE;
				END_IF;
			END_IF;

		eOPMAINT:	(*Maintenance -------------------------------------*)
			IF sI_CleanDevCmd.bInit THEN
				fO_TargetPosition := fI_ServicePosition;
				bL_MotionActive   := TRUE;
				bL_AxisReady      := FALSE;

			ELSIF sI_CleanDevCmd.bPrep THEN
				bL_MotionActive   := FALSE;
				bL_AxisReady      := TRUE;

			ELSIF sI_CleanDevCmd.bStart THEN
				bL_MotionActive   := FALSE;
				bL_AxisReady      := TRUE;

			ELSIF sI_CleanDevCmd.bStop THEN
				bL_MotionActive   := FALSE;
				bL_AxisReady      := TRUE;

			ELSE	(*Command removed, wait until axis finished movement*)
				IF NOT bL_MoveDone THEN
					bL_MotionActive := TRUE;
					bL_AxisReady    := FALSE;
				ELSE
					bL_MotionActive := FALSE;
					bL_AxisReady    := TRUE;
				END_IF;
			END_IF;

		eOPSHUTTEROPEN: (*Open Shutters, do nothing*)
			bL_AxisReady    := TRUE;
			bL_MotionActive := FALSE;

		ELSE
			bL_MotionActive := FALSE;
			bL_AxisReady    := TRUE;
		END_CASE;

		(*In case of abort set target position to current position and wait for MoveDone flag*)
		IF sI_CleanDevCmd.bAbort THEN
			fO_TargetPosition := fI_CurrentPosition;
		END_IF;

ELSE		(* MANUAL MODE *)
	IF sI_ManualCommands.bI_Do AND NOT sI_ManualCommands.bI_Undo THEN
		fO_TargetPosition := sI_ManualCommands.fI_Start_position;
		bL_AxisReady      := FALSE;
	ELSIF NOT sI_ManualCommands.bI_Do AND sI_ManualCommands.bI_Undo THEN
		fO_TargetPosition := sI_ManualCommands.fI_Stop_position;
		bL_AxisReady      := FALSE;
	ELSE
		bL_AxisReady      := TRUE;
		fO_TargetPosition := fI_CurrentPosition;
	END_IF;

	bL_MotionActive := sI_ManualCommands.bI_Do OR sI_ManualCommands.bI_Undo;
END_IF;
END_ACTION

END_FUNCTION_BLOCK

// ---- POUs/Machine/CleaningStation/FB_SHUTTER.TcPOU
FUNCTION_BLOCK FB_SHUTTER

(******************************************************************************************)
(*	FILENAME:	FB_SHUTTER											*)
(*	PROJECT:	Steinemann											*)
(*	COPYRIGHT:	Wifag-Polytype								*)
(*	ENVIRONMENT:	TwinCat2, v2.11							*)
(*	VERSION:	1.0															*)
(*	DESCRIPTION:															*)
(*		This function controls the shutters 		*)
(*	AUTHOR:	FAF							*)
(*																*)
(******************************************************************************************)
(*	Changes:													*)
(******************************************************************************************)
(*	Date	Authtor	Descriptons									*)
(*																*)
(******************************************************************************************)
VAR_INPUT
	(*From Shutter*)
	bI_ShutterInletClosed		: BOOL;
	bI_ShutterOutletClosed	: BOOL;

	(*From Machine*)
	bI_ESTopOk				: BOOL;	(*General ready flag*)

	(*Commands from Cleaning Process Controller*)
	sI_CleanDevCmd				: ST_CLEANING_DEV_CMD;	(*Initialize operation*)

	(*From User*)
	bI_ForceInletOpen			: BOOL;
	bI_ForceInletClose		: BOOL;
	bI_ForceOutletOpen		: BOOL;
	bI_ForceOutletClose		: BOOL;

	pC_MsgInterface		: POINTER TO ST_ADS_MSG_IF;
	iC_BlockId				: INT;
END_VAR

VAR_OUTPUT
	(*To Shutter*)
	bO_ShutterInletOpen		:BOOL;
	bO_ShutterInletClose	:BOOL;
	bO_ShutterOutletOpen	:BOOL;
	bO_ShutterOutletClose	:BOOL;

	(*To machine/user*)
	bO_SafetyOk				: BOOL;	(*Safety ok for movement*)
	sO_CleanDevStatus	:ST_CLEANING_DEV_STATUS;	(*Initialize operation*)
END_VAR

VAR
	cL_State									:	BYTE := cL_UNKNOWN;	(*State type*)
	tL_OpenTime								: TON;			(* Timer for Sensor check *)
	bL_AxisReady							: BOOL := FALSE;
	bL_CloseRequest						: BOOL := FALSE;
	bL_OpenRequest						: BOOL := FALSE;
	bL_SafeRunningCondition		: BOOL := FALSE;
	bL_RefKnown								: BOOL := FALSE;
	bL_AllShutterClosed				: BOOL;

	bL_ShutterInletOpen				: BOOL;
	bL_ShutterInletClose			: BOOL;
	bL_ShutterOutletOpen			: BOOL;
	bL_ShutterOutletClose			: BOOL;

	fB_Motor_Switch_A					: FB_MOTOR_SWITCH;
	fB_Motor_Switch_B					: FB_MOTOR_SWITCH;

	(*Message Queue*)
(* 	fB_MsgQueue				          		: FB_MSG_QUEUE;
	fB_MsgHandler										: FB_MSG_HANDLER;
	sL_MsgConfig										: ST_MSG_CONFIG;
	fB_Msg													: ARRAY [1..iC_NUM_MSG] OF FB_MESSAGE;*)
END_VAR

VAR CONSTANT
	(*State*)
	cL_OPEN						: BYTE := 01;										(*Shutter open = Safety not ok*)
	cL_CLOSING				: BYTE := 12;										(*Shutter moving = Safety not ok*)
	cL_CLOSED					: BYTE := 02;										(*Shutter closed = Safety ok*)
	cL_OPENING				: BYTE := 21;										(*Shutter moving = Safety not ok*)
	cL_UNKNOWN				: BYTE := 99;										(*State unknown, Init*)

	iC_NUM_MSG											: INT :=1;
END_VAR

(*----------------------------------------------------------------------------------------------------------------------------------------------- *)
(*Running Conditions *)
(*----------------------------------------------------------------------------------------------------------------------------------------------- *)
IF bI_ESTopOk THEN
	bL_SafeRunningCondition := TRUE;
ELSE
	bL_SafeRunningCondition := FALSE;
END_IF;

bL_AllShutterClosed := bI_ShutterInletClosed AND bI_ShutterOutletClosed;

(*----------------------------------------------------------------------------------------------------------------------------------------------- *)
(* Motion Control  *)
(*----------------------------------------------------------------------------------------------------------------------------------------------- *)
IF bL_RefKnown = FALSE THEN	(* Startup condition*)
	bL_OpenRequest := FALSE;

	IF bL_AllShutterClosed THEN		(**)
		bL_CloseRequest := FALSE;
		bL_RefKnown     := TRUE;
	ELSE
		bL_CloseRequest := TRUE;
		bL_RefKnown     := FALSE;
	END_IF;																(**)
ELSE	(* Axis has been initialized *)
	IF sI_CleanDevCmd.bService THEN
		ServiceMode();
	ELSE
		bL_OpenRequest	:= FALSE;
		bL_CloseRequest := FALSE;
	END_IF;
END_IF;

IF bL_SafeRunningCondition THEN
	ShutterProcess();
ELSE
	bL_ShutterInletOpen   := FALSE;
	bL_ShutterInletClose  := FALSE;
	bL_ShutterOutletOpen  := FALSE;
	bL_ShutterOutletClose := FALSE;
	bL_AxisReady          := FALSE;
END_IF;

(*----------------------------------------------------------------------------------------------------------------------- *)
(* Output Structure Data Update  																																													*)
(*----------------------------------------------------------------------------------------------------------------------- *)
sO_CleanDevStatus.bBusy     := NOT(bL_AxisReady) AND bL_SafeRunningCondition;
sO_CleanDevStatus.bReady    := bL_AxisReady;
sO_CleanDevStatus.bRefKnown := bL_RefKnown;
sO_CleanDevStatus.bError    := FALSE;

(*----------------------------------------------------------------------------------------------------------------------- *)
(* Safety																																													                        *)
(*----------------------------------------------------------------------------------------------------------------------- *)
IF bL_AllShutterClosed THEN
	bO_SafetyOk := TRUE;
ELSE
	bO_SafetyOk := FALSE;
END_IF;

fB_Motor_Switch_A.bI_A := bL_ShutterInletClose;
fB_Motor_Switch_A.bI_B := bL_ShutterInletOpen;

fB_Motor_Switch_A();

bO_ShutterInletClose := fB_Motor_Switch_A.bO_QA;
bO_ShutterInletOpen  := fB_Motor_Switch_A.bO_QB;

fB_Motor_Switch_B.bI_A := bL_ShutterOutletClose;
fB_Motor_Switch_B.bI_B := bL_ShutterOutletOpen;

fB_Motor_Switch_B();

bO_ShutterOutletClose := fB_Motor_Switch_B.bO_QA;
bO_ShutterOutletOpen  := fB_Motor_Switch_B.bO_QB;

(*----------------------------------------------------------------------------------------------------------------------- *)
(*--------------------------------- Fault Diagnosis and Management  ---------------------------------- *)
(*----------------------------------------------------------------------------------------------------------------------- *)
(*fB_Msg[1](bI_Status:=NOT bO_SafetyOk);

fB_MsgQueue(); *)

ACTION ServiceMode:
(*Mode selection*)
IF sI_CleanDevCmd.bAuto THEN	(*Control by cleaning process*)
	CASE 	sI_CleanDevCmd.eOperation OF
		eNOP:	(*No operation active*)
			bL_OpenRequest				:= FALSE;
			bL_CloseRequest 			:= FALSE;
		eOPCLEAN, eOPCAPENTER, eOPCAPEXIT, eOPPURGE, eOPPREPSERVICE, eOPENDSERVICE, eOPSTARTUP:	(*All modes except maintenance and shutter open*)
			IF sI_CleanDevCmd.bInit THEN
				bL_CloseRequest 		:= TRUE;
				bL_OpenRequest			:= FALSE;
			ELSE
				bL_OpenRequest			:= FALSE;
				bL_CloseRequest 		:= FALSE;
			END_IF;

		eOPMAINT:	(*Maintenance -------------------------------------*)
			IF sI_CleanDevCmd.bInit THEN
				bL_CloseRequest 		:= TRUE;
				bL_OpenRequest			:= FALSE;
			ELSIF sI_CleanDevCmd.bStart THEN
				bL_CloseRequest 		:= FALSE;
				bL_OpenRequest			:= TRUE;
			ELSE
				bL_OpenRequest			:= FALSE;
				bL_CloseRequest 		:= FALSE;
			END_IF;

		eOPSHUTTEROPEN:	(*Open Shutter ------------------------------*)
			IF sI_CleanDevCmd.bStart THEN
				bL_CloseRequest 		:= FALSE;
				bL_OpenRequest			:= TRUE;
			ELSE
				bL_OpenRequest			:= FALSE;
				bL_CloseRequest 		:= FALSE;
			END_IF;
		ELSE
			bL_OpenRequest				:= FALSE;
			bL_CloseRequest 			:= FALSE;
		END_CASE;

ELSE		(* MANUAL MODE *)
	bL_OpenRequest			:= FALSE;
	bL_CloseRequest 		:= FALSE;
END_IF;
END_ACTION

ACTION ShutterProcess:
(*Default*)

(*Mode selection*)
IF sI_CleanDevCmd.bAuto THEN	(*Control by cleaning process*)
	IF NOT bL_RefKnown THEN
		cL_State:= cL_UNKNOWN;
	END_IF;
	
	(*State Machine -----------------------------------------------------------------*)
	CASE cL_State OF
		cL_UNKNOWN:
			IF bL_AllShutterClosed THEN
				cL_State:= cL_CLOSED;
			ELSE
				cL_State:= cL_UNKNOWN;
			END_IF;
	
			bL_AxisReady:=FALSE;
			bL_ShutterInletOpen	:=FALSE;
			bL_ShutterOutletOpen:=FALSE;
			bL_ShutterInletClose:=bL_CloseRequest AND NOT bI_ShutterInletClosed;
			bL_ShutterOutletClose:=bL_CloseRequest AND NOT bI_ShutterOutletClosed;
	
		cL_OPEN:
			IF bL_CloseRequest THEN
				cL_State:= cL_CLOSING;
				bL_AxisReady:=FALSE;
			ELSE
				cL_State:= cL_OPEN;
				bL_AxisReady:=TRUE;
			END_IF;
	
			tL_OpenTime.IN:=FALSE;
			bL_ShutterInletOpen	:=FALSE;
			bL_ShutterOutletOpen:=FALSE;
			bL_ShutterInletClose:=FALSE;
			bL_ShutterOutletClose:=FALSE;
	
		cL_CLOSING:
			IF bL_AllShutterClosed THEN
				cL_State:= cL_CLOSED;
			ELSE
				cL_State:= cL_CLOSING;
			END_IF;
	
			tL_OpenTime.IN:=FALSE;
			bL_ShutterInletOpen	:=FALSE;
			bL_ShutterOutletOpen:=FALSE;
			bL_ShutterInletClose:= NOT bI_ShutterInletClosed;
			bL_ShutterOutletClose:=NOT bI_ShutterOutletClosed;
			bL_AxisReady:=FALSE;
	
		cL_CLOSED:
			IF bL_OpenRequest THEN
				cL_State:= cL_OPENING;

				tL_OpenTime.IN:=TRUE;
				tL_OpenTime.PT:=T#20s;
				bL_AxisReady:=FALSE;
			ELSE
				cL_State:= cL_CLOSED;
				tL_OpenTime.IN:=FALSE;
				bL_AxisReady:=TRUE;
			END_IF;
	
			bL_ShutterInletOpen	:=FALSE;
			bL_ShutterOutletOpen:=FALSE;
			bL_ShutterInletClose:=TRUE;
			bL_ShutterOutletClose:=TRUE;

		cL_OPENING:
			IF tL_OpenTime.Q THEN
				cL_State:= cL_OPEN;
				tL_OpenTime.IN:=FALSE;
			ELSE
				tL_OpenTime.IN:=TRUE;
				cL_State:= cL_OPENING;
			END_IF;

			bL_ShutterInletOpen	:=TRUE;
			bL_ShutterOutletOpen:=TRUE;
			bL_ShutterInletClose:=FALSE;
			bL_ShutterOutletClose:=FALSE;
			bL_AxisReady:=FALSE;
	END_CASE;
	tL_OpenTime();
ELSE		(* MANUAL MODE *)
			bL_ShutterInletOpen	:=bI_ForceInletOpen;
			bL_ShutterOutletOpen:=bI_ForceOutletOpen;
			bL_ShutterInletClose:=bI_ForceInletClose;
			bL_ShutterOutletClose:=bI_ForceOutletClose;
END_IF;
END_ACTION

END_FUNCTION_BLOCK

// ---- POUs/Machine/EffectiveEncoderResolutionDetection/FB_EffectiveEncoderResolutionDetection.TcPOU
FUNCTION_BLOCK FB_EffectiveEncoderResolutionDetection EXTENDS FB_Commons
VAR_INPUT
  (*EL1252*)
  bIKp_MarkTrigger01    AT%I* : BOOL;        // First  mark sensor - Trigger
  tIKp_TimeStampPos01   AT%I* : T_DCTIME64;  // First  mark sensor - RisingEdge  @EL1252
  tIKn_TimeStampNeg01   AT%I* : T_DCTIME64;  // First  mark sensor - FallingEdge @EL1252
  bIKp_MarkTrigger02    AT%I* : BOOL;        // Second mark sensor - Trigger
  tIKp_TimeStampPos02   AT%I* : T_DCTIME64;  // Second mark sensor - RisingEdge  @EL1252
  tIKn_TimeStampNeg02   AT%I* : T_DCTIME64;  // Second mark sensor - FallingEdge @EL1252
  nPulse                      : DINT;        // encoder pulse input
  nDisInPulseFilterSz         : UDINT;       // mav filter size for measured distance in encoder steps (from machine) 
    
  // settings
  fCurrentResolution          : LREAL;       // current used resolution (given from machine), encoder step size
  fEncoderPulseDistMin        : LREAL;       // [pulse] defines the min sensor distance in pulse, range minimum
  fEncoderPulseDistMax        : LREAL;       // [pulse] defines the max sensor distance in pulse, range maximum
  fMinMarkLength              : LREAL:=2000; // [um] minimal mark lenght to accept a measurement
  fMaxMarkLength              : LREAL:=6000; // [um] maximal mark lenght to accept a measurement
END_VAR
VAR_OUTPUT
  bUpdate                     : BOOL;        // a valid new measurment
  fDisInPulse                 : LREAL;       // disntance in encoder pulse
END_VAR
VAR
  bInitOk                     : BOOL;        // initialized
   
  fSpeedPulse                 : LREAL;       // current encoder speed [pulse/s]
  fSpeedUm_s                  : LREAL;       // current speed [um/s]
  fbMark1,fbMark2             : RF_TRIG;     // edge detection
  bMeasurementActive          : BOOL;        // a measurement started
  bS1_MarkStarted, bS2_MarkStarted : BOOL;
  nMeasurementCounter         : UDINT;       // counter for measurements
  nCurrentDistActive          : DINT;        // current distance during active measurement
  bVerbose                    : BOOL;
  // errors
  bLower, bHigher, bAborted   : BOOL;        // ui errors
  bMarkInvalidLength_S1, bMarkInvalidLength_S2 : BOOL; // detected marks too short or too long
  nMarkLength_S1, nMarkLength_S2 : UDINT;    // mark length measured in [um]
  
  // time calculations
  tNowDc                      : T_DCTIME64;  // Get Current Timestamp (now
  _fCycleTime                 : LREAL;       // Current cycle time [s]

  // position
  fDistMeasured               : LREAL;       // distance measured [pulse]
  fbFilterMavDisInPulse       : FB_FILTER_MAV; // Moving everage filter
  //fbFilterMavSpeed            : FB_FILTER_MAV; // Moving everage filter
  fAbortDistUm                : LREAL;
  
  // helper measurement
  nPosStart, nPosEnd : DINT;                 // encoder positions detectec (exact by trigger, timestamp and speed based approximation)
  nPosFalling1, nPosFalling2 : DINT;         // exact position in [pulse]
  bRising_S1, bFalling_S1, bRising_S2, bFalling_S2 : BOOL;    // sensor edge detection

END_VAR
VAR CONSTANT
  nC_MinMarkLength            : LREAL := 2_000; // min. mark length in [um]
END_VAR

// check & correct parameter
IF NOT bInitOk THEN RETURN; END_IF;

bUpdate := FALSE;

// time caluclations
tNowDc := F_GetCurDcTaskTime64();                  // current dc time (most accurate time stamp we have)
_fCycleTime := calcCycleTime(tCurrent:=tNowDc);     // calculate cycle time of this fb

// input edge detection
fbMark1(CLK:=bIKp_MarkTrigger01);
fbMark2(CLK:=bIKp_MarkTrigger02);

// track position & speed
position(
  fResolutionInput:=fCurrentResolution, 
  lPosReference:=nPulse, 
  fMasterSpeed=>fSpeedUm_s,    // [um/s]
  fPulseSpeed=>fSpeedPulse,    // [p/s]
);

measure(bUpdate=>bUpdate, fEncoderDistance=>fDistMeasured);
IF bUpdate THEN
  // check range (given from machine)
  bHigher := SEL(fDistMeasured > fEncoderPulseDistMax, FALSE, TRUE);  IF bVerbose AND bHigher THEN LogWarning('Measured distance in pulse LONGER than max range'); END_IF
  bLower  := SEL(fDistMeasured < fEncoderPulseDistMin, FALSE, TRUE);  IF bVerbose AND bLower  THEN LogWarning('Measured distance in pulse SHORTER than min range'); END_IF

  IF NOT bHigher AND NOT bLower THEN  
    // measurement ok
    fbFilterMavDisInPulse(fI_Input:=fDistMeasured, iI_NbInputs:=TO_UINT(LIMIT(1, nDisInPulseFilterSz, fbFilterMavDisInPulse.cL_BUFFER_MAX))); // moving average filter
    fDisInPulse := fbFilterMavDisInPulse.fO_OutputMav;
  END_IF
  
  nMeasurementCounter := (nMeasurementCounter + 1) MOD 1000;  // limit to 0-1000
END_IF

// 
METHOD PRIVATE abortMarkEndSearch : BOOL
VAR_INPUT
  nStart  : DINT;     // pulse
  nEnd    : DINT;     // pulse
END_VAR
VAR
  nDist   : DINT;     // [pulse]
  fDistUm : LREAL;    // um
END_VAR
// pulse elapsed * resolution [um/pulse] => pos in [um]
nDist := ABS(nEnd - nStart);    // distance in pulse (1-2 cycle too late)
fDistUm := nDist * fCurrentResolution;   // distance in [um]  

fAbortDistUm := fMaxMarkLength + (2*_fCycleTime * fSpeedUm_s);

abortMarkEndSearch := fDistUm > fAbortDistUm;
END_METHOD

METHOD PRIVATE calcCycleTime : LREAL
VAR_INPUT
  tCurrent : T_DCTIME64;
END_VAR
VAR_INST
  tLastTimeStamp : T_DCTIME64 := 0;
END_VAR
calcCycleTime := (TO_LREAL(tCurrent) - TO_LREAL(tLastTimeStamp)) * 1E-9;
tLastTimeStamp  := tCurrent;  // memory timestamp
END_METHOD

METHOD PRIVATE checkMarkLength : BOOL
VAR_INPUT
  nRef : DINT;     // pulse
  nOther : DINT;   // pluse
END_VAR
VAR_OUTPUT
  nLen : DINT;     // mark length in pulse
END_VAR
VAR
  fMarkLen : LREAL;  // [um]
END_VAR
IF fCurrentResolution = 0 THEN RETURN; END_IF

// pulse elapsed * resolution [pulse/um] => pos in [um]
nLen := ABS(nOther - nRef);
fMarkLen := nLen * fCurrentResolution;
IF fMarkLen > fMinMarkLength AND fMarkLen < fMaxMarkLength THEN
  // mark within spec
  checkMarkLength := TRUE;
  IF bVerbose THEN LogInfo(F_Concat3('Mark length= ', TO_STRING(fMarkLen), 'um')); END_IF
ELSE
  IF bVerbose THEN LogWarning(F_Concat5('Mark length invalid: ', TO_STRING(fMarkLen), 'um', ' too short or too long', '')); END_IF
END_IF
END_METHOD

METHOD PRIVATE getExactPosition : DINT
VAR_INPUT
  tNow : T_DCTIME64;    // current system time
  nPos : DINT;          // current (encoder) position at the current timestamp
  tEdge : T_DCTIME64;   // detected time
  fSpeed : LREAL;       // current speed
END_VAR
VAR
  fCurrentTimeStamp : LREAL;
  fSensor_TimeStamp : LREAL;
  fDeltaDistance    : LREAL;      // Distance that the substrate moved between the detection and the treatment of the information
END_VAR
IF fCurrentResolution = 0 THEN RETURN; END_IF

// Calculate the original position in our position domain
fCurrentTimeStamp  := (ULINT_TO_LREAL(tNow) - (GVL_WEU.nC_CurrentTimeStampComp * 1_000)) / 1_000_000.0; // [ms]
fSensor_TimeStamp := (ULINT_TO_LREAL(tEdge) - (GVL_WEU.nC_SensorTimeStampComp  * 1_000)) / 1_000_000.0; // [ms]

// Treatment of the information
fDeltaDistance   := (fCurrentTimeStamp - fSensor_TimeStamp) * 0.001 * fSpeed;	      // Distance in pulses that the substrate has traveled between the sensor detection and the PLC treatment
// not conversion to px   nDeltaPosition := FC_LREAL_TO_DINT(fDeltaDistance * (1 / (0.0254 / fCurrentResolution)));   // 1/1px	(* Travel of the substrate between the time of acquisition and the time of treatment
getExactPosition := FC_LREAL_TO_DINT(TO_LREAL(nPos) - fDeltaDistance);
END_METHOD

METHOD Init
Reset();

bInitOk := TRUE;
END_METHOD

METHOD PRIVATE measure
VAR_OUTPUT
  bUpdate : BOOL;
  fEncoderDistance : LREAL;
END_VAR
bUpdate := FALSE;
bRising_S1 := fbMark1.RT;
bRising_S2 := fbMark2.RT;
bFalling_S1 := fbMark1.FT;    // wait on falling edge always 
bFalling_S2 := fbMark2.FT;

IF NOT bMeasurementActive THEN
  
  //-- S1 sensor evaluation (no measurement is active)
  // rising
  IF bRising_S1 AND NOT bS1_MarkStarted THEN
    nPosStart := getExactPosition(tNow:=tNowDc, nPos:=nPulse, tEdge:=tIKp_TimeStampPos01, fSpeed:=fSpeedPulse);
    bS1_MarkStarted := TRUE;
    bAborted := FALSE; bMarkInvalidLength_S1 := FALSE; bMarkInvalidLength_S2 := FALSE;
  END_IF

  // falling (after rising)
  IF bFalling_S1 AND bS1_MarkStarted THEN
    bS1_MarkStarted := FALSE;           // mark done
    nPosFalling1 := getExactPosition(tNow:=tNowDc, nPos:=nPulse, tEdge:=tIKn_TimeStampNeg01, fSpeed:=fSpeedPulse);
  
    IF checkMarkLength( nRef := nPosStart, nOther := nPosFalling1) THEN
      bMeasurementActive := TRUE;           // start measurement after rising&falling edge
    ELSE
      bMarkInvalidLength_S1 := TRUE;
    END_IF

  // abort mark if no falling given
  ELSIF bS1_MarkStarted AND abortMarkEndSearch(nStart:=nPosStart, nEnd:=nPulse) THEN  // abort if max mark length exeeded
    bS1_MarkStarted := FALSE;         // mark done
    bMarkInvalidLength_S1 := TRUE;    // mark end missed (too long?)
    IF bVerbose THEN LogWarning('S1 mark missing end, mark too long, ignore mark'); END_IF
  END_IF
  
ELSE
  
  //-- S2 Second Sensor (Stop) evaluation when measurement is active
  //   only when measurement started and rising within range
  IF (nPulse - nPosStart) >= fEncoderPulseDistMin THEN                  // bigger than minimum pulse (enable sensor 2 detection)
    // rising
    IF bRising_S2 AND NOT bS2_MarkStarted THEN 
      nPosEnd := getExactPosition(tNow:=tNowDc, nPos:=nPulse, tEdge:=tIKp_TimeStampPos02, fSpeed:=fSpeedPulse);    
      bAborted := FALSE; bMarkInvalidLength_S2 := FALSE;
      bS2_MarkStarted := TRUE;  
    END_IF
    
    // falling
    IF bFalling_S2 AND bS2_MarkStarted THEN
      bS2_MarkStarted := FALSE;
      nPosFalling2 := getExactPosition(tNow:=tNowDc, nPos:=nPulse, tEdge:=tIKn_TimeStampNeg02, fSpeed:=fSpeedPulse);  
      
      IF checkMarkLength( nRef := nPosEnd, nOther := nPosFalling2) THEN
        bUpdate := TRUE;
        bMeasurementActive := FALSE;      // stop measurement
      ELSE
        bMarkInvalidLength_S2 := TRUE;
      END_IF

    // abort mark if no falling given
    ELSIF bS2_MarkStarted AND abortMarkEndSearch(nStart:=nPosEnd, nEnd:=nPulse) THEN  // abort if max mark length exeeded
      bS1_MarkStarted := FALSE;         // mark done
      bMarkInvalidLength_S2 := TRUE;    // mark end missed (too long?)
      IF bVerbose THEN LogWarning('S2 mark missing end, mark too long, ignore mark'); END_IF
    END_IF
  
  // abort measurement, no valid mark within max pulse distance
  //       TODO: the nPulse can be 1-2 cycle later than the nPosStart so maybe we should add a marging here to fEncoderPulseDistMax + 1 cycle
  ELSIF ( (nPulse - nPosStart) > (fEncoderPulseDistMax) ) THEN    // bigger than maximum pulse (disable sensor 2 and abort measurement)
    IF bVerbose THEN LogWarning('S2 mark detected too far , ignore measurement'); END_IF
    bAborted := TRUE;                   // abort measurement
    bMeasurementActive := FALSE;        // abort measurement
    bS2_MarkStarted := FALSE;           // mark done
  
  // invalid speed (machine stopped while measuring) ignore any triggers
  ELSIF fSpeedPulse = 0 THEN
    bS1_MarkStarted := bS2_MarkStarted := FALSE;
    bMeasurementActive := FALSE;
	END_IF
  
END_IF

// debug current distance (view)
IF bMeasurementActive THEN nCurrentDistActive := (nPulse - nPosStart); END_IF 

// valid measurment -> update output
IF bUpdate THEN
  fEncoderDistance := nPosEnd-nPosStart;
END_IF
END_METHOD

METHOD PRIVATE position
VAR_INPUT
  lPosReference         : DINT;			                (*Position reference pulse count in [pulse (resolution)]*)
  fResolutionInput      : LREAL := 1;	              (*Encoder resolution in [um/increment]*)
END_VAR
VAR_OUTPUT
  fMasterPosition       : LREAL;                    (*Master position in [um]*)
  fPulsePosition        : LREAL;
  fMasterSpeed          : LREAL;                    (*Master speed in [um/s]*)
  fPulseSpeed           : LREAL;                    (*Pulse speed*)
END_VAR
VAR_INST
  bReset : BOOL;

  lL_Reference_Reg       : DINT := 0;               (*Position reference pulse count register [pulse (resolution)]*)
  fL_Master_Position_Reg : LREAL := 0;	            (*Master position register (last position) [um]*)
  fL_Pulse_Position_Reg  : LREAL := 0;	            (*Master position register (last position) [?]*)
  lL_Delta               : DINT;                    (*Delta of position reference pulses*)
  fDelta : LREAL;
  fb_MavDelta            : FB_FILTER_MAV;           (*Moving everage filter*)

  fL_MasterSpeed_reg     : LREAL;                   (*Speed register [m/s]*)
  fL_PulseSpeed_reg      : LREAL;                   (*Speed [p/s]*)
END_VAR
VAR CONSTANT
  iC_FilterDepth         : UINT := 1;                (*Default filter depth*)
  fC_MinSpeed            : LREAL := 0.02;            (*min speed [m/s]*)
END_VAR
IF _fCycleTime = 0 THEN RETURN; END_IF
IF bReset THEN bReset := FALSE;
  lL_Reference_Reg := lPosReference;
  fL_Master_Position_reg := 0; fL_Pulse_Position_Reg := 0;
  fL_MasterSpeed_reg := 0; fL_PulseSpeed_reg := 0;
END_IF 

lL_Delta:=(lPosReference-lL_Reference_Reg);  // DINT because diff correct on wrap over
// filter
fb_MavDelta.fI_Input    := DINT_TO_LREAL(lL_Delta);       // encoder signal jitter filter
fb_MavDelta.iI_NbInputs := iC_FilterDepth;
fb_MavDelta();
fDelta := TO_LREAL(lL_Delta);    //fb_MavDelta.fO_OutputMav  (filtered)

// Position & Speed Calculation 
fMasterPosition := fDelta * fResolutionInput + fL_Master_Position_Reg;
fPulsePosition  := fDelta * 1 + fL_Pulse_Position_Reg;

(*Speed Calculation*)
fMasterSpeed := (fMasterPosition - fL_Master_Position_Reg) * (1 / _fCycleTime);  // um/s      // * 0.000001 um -> m 
IF LrealIsNaN(x:=fMasterSpeed) THEN fMasterSpeed := fL_MasterSpeed_reg; END_IF
fPulseSpeed  := (fPulsePosition - fL_Pulse_Position_Reg) * (1 / _fCycleTime); // * 0.000001;  // um -> 
IF LrealIsNaN(x:=fPulseSpeed) THEN fPulseSpeed := fL_PulseSpeed_reg; END_IF

(*Update Registers*)
lL_Reference_Reg       := lPosReference;
fL_Master_Position_Reg := fMasterPosition; fL_Pulse_Position_Reg := fPulsePosition;
fL_MasterSpeed_reg     := fMasterSpeed; fL_PulseSpeed_reg := fPulseSpeed;
END_METHOD

METHOD PRIVATE Reset
nMeasurementCounter := 0;
END_METHOD

END_FUNCTION_BLOCK

// ---- POUs/Machine/ExhaustSystem/FB_ExhaustSystemPrint.TcPOU
FUNCTION_BLOCK FB_ExhaustSystemPrint
VAR_INPUT
  bI_FUReady                         AT %I* : BOOL;   (*FU ready*)
  iI_VacuumMeasurement               AT %I* : UINT;   (*Analog input: vacuum measurement*)
  bPrintActive                              : BOOL;   (*Printing active*)
END_VAR

VAR_OUTPUT
  bO_FUActivate                      AT %Q* : BOOL;   (*FU activation*)
  OnExhaustSetpoint                  AT %Q* : UINT;   (*Analog output: pump setpoint*)

  bExhaustError                             : BOOL;   (*Exhaust system ok and ready*)
  // detailed status (for messages)
  bFUReady                                  : BOOL;   (*FU ready*)
  bVacuumWarningLevel                       : BOOL;   (*Vacuum warning level reached*)
  bVacuumErrorLevel                         : BOOL;   (*Vacuum error level reached*)
END_VAR

VAR
  iL_Counter                                : INT;    (*Basic counter*)
  bMappingChecked                           : BOOL;   (*Checked mapped variable status*)
  bMapping_FUReady_Done                     : BOOL;   (*FUReady is mapped*)
  
  fb_TofFUOffDelay                          : TOF;    (*FU off delay*)
  fb_TonVacuumCheckDelay                    : TON;    (*Vacuum check delay*)

  fL_VacuumAnalogLevelMBar                  : REAL;   (*Actual value analog-input in mBar*)
END_VAR

VAR PERSISTENT
  tR_FUOffDelay                             : TIME := T#3M;   (*FU off delay time*)
  tR_VacuumCheckDelay                       : TIME := T#10S;  (*Vacuum check delay time*)

  iR_VacuumAnalogMinDigit                   : UINT := 0;      (*Min value analog-input in digit*)
  iR_VacuumAnalogMaxDigit                   : UINT := 32767;  (*Max value analog-input in digit*)
  fR_VacuumAnalogMinMBar                    : REAL := 0;      (*Min value analog-input in mBar*)
  fR_VacuumAnalogMaxMBar                    : REAL := 50.0;   (*Max value analog-input in mBar*)
  fR_VacuumWarningLevelMBar                 : REAL := 20.0;   (*Warning level in mBar*)
  fR_VacuumErrorLevelMBar                   : REAL := 10.0;   (*Error level in mBar*)

  iR_VacuumPumpSetPercent                   : UINT := 0;      (*Pump setpoinr [%]*)
  iR_VacuumPumpSetpointMaxDigit             : UINT := 13762;  (*Max value analog-output in digit, max pump = 4.2V*)
END_VAR

// mapping check
IF NOT bMappingChecked THEN checkMapping(); END_IF
IF NOT bMapping_FUReady_Done THEN bI_FUReady := TRUE; END_IF    // if not mapped is ready


bFUReady := bI_FUReady;  // AND bO_FUActivate?

fb_TofFUOffDelay(IN := bPrintActive, PT := tR_FUOffDelay);    // turn-off delay
bO_FUActivate := fb_TofFUOffDelay.Q;

fL_VacuumAnalogLevelMBar := UINT_TO_REAL(iI_VacuumMeasurement) * fR_VacuumAnalogMaxMBar / iR_VacuumAnalogMaxDigit;

fb_TonVacuumCheckDelay(IN := bO_FUActivate, PT := tR_VacuumCheckDelay);   // delay for vacum measurement
IF fb_TonVacuumCheckDelay.Q THEN
  // check levels and set waring/error
  bVacuumWarningLevel := fL_VacuumAnalogLevelMBar < fR_VacuumWarningLevelMBar;
  bVacuumErrorLevel   := fL_VacuumAnalogLevelMBar < fR_VacuumErrorLevelMBar;
END_IF


bExhaustError := NOT bFUReady OR (bVacuumErrorLevel AND bO_FUActivate);

OnExhaustSetpoint := REAL_TO_UINT(UINT_TO_REAL(iR_VacuumPumpSetpointMaxDigit) / 100 * iR_VacuumPumpSetPercent);

METHOD PRIVATE checkMapping
VAR_INPUT
END_VAR
bMapping_FUReady_Done := F_GetMappingStatus(p:=ADR(bI_FUReady), n:=SIZEOF(bI_FUReady)) > EPlcMappingStatus.MS_Unmapped;

bMappingChecked := TRUE;
END_METHOD

METHOD mAckError : BOOL
VAR_INPUT
END_VAR
bVacuumWarningLevel := FALSE;
bVacuumErrorLevel   := FALSE;
END_METHOD

END_FUNCTION_BLOCK

// ---- POUs/Machine/FB_FILTER_MAV_1000.TcPOU
FUNCTION_BLOCK FB_FILTER_MAV_1000
(*************************************************************************************************)
(*  FILENAME:    FB_FILTER_MAV_1000.EXP                                                          *)
(*  PROJECT:     CALMAR PUPLC                                                                    *)
(*  COPYRIGHT:   All rights reserved (c) Wifag//Polytype, Fribourg/Switzerland (2016)            *)
(*  ENVIRONMENT: TwinCAT PLC                                                                     *)
(*  VERSION:     <version>                                                                       *)
(*************************************************************************************************)
(*  DESCRIPTION:                                                                   <description> *)
(*     Moving everage filter.                                                                    *)
(*                                                                                </description> *)
(*************************************************************************************************)

VAR_INPUT
  fI_Input                  : LREAL;                              (*Input value*)
  iI_NbInputs               : UINT;                               (*Number of inputs*)

  bI_Reset                  : BOOL;                               (*Reset function*)
END_VAR

VAR_OUTPUT
  fO_OutputMav              : LREAL;                              (*Output filtered value*)
END_VAR

VAR
  bL_Init                   : BOOL;                               (*Init function*)
  fL_Buffer                 : ARRAY [1..cL_BUFFER_MAX] OF LREAL;  (*Buffer for values*)
  fL_Sum                    : LREAL;                              (*Sum of values*)

  iL_Counter                : INT;                                (*Internal counter*)
  iL_Counter2               : INT;                                (*Internal counter*)
END_VAR

VAR CONSTANT
  cL_BUFFER_MAX             : UINT := 1000;                       (*Const buffer max size*)
END_VAR

IF (iI_NbInputs = 0) OR (iI_NbInputs > cL_BUFFER_MAX) THEN
  iI_NbInputs := cL_BUFFER_MAX;
END_IF

IF NOT bL_Init OR bI_Reset THEN
  bL_Init := TRUE;

  FOR iL_Counter := 1 TO UINT_TO_INT(iI_NbInputs) DO
    fL_Buffer[iL_Counter] := fI_Input;
  END_FOR

  fO_OutputMav := fI_Input;
ELSE
  iL_Counter := iL_Counter + 1;
  IF iL_Counter > UINT_TO_INT(iI_NbInputs) THEN
    iL_Counter := 1;
  END_IF

  fL_Buffer[iL_Counter] := fI_Input;

  
  fL_Sum := 0;
  FOR iL_Counter2 := 1 TO UINT_TO_INT(iI_NbInputs) DO
    fL_Sum := fL_Sum + fL_Buffer[iL_Counter2];
  END_FOR
  fO_OutputMav := fL_Sum / iI_NbInputs;
END_IF;

(********************************* END OF FB *****************************************************)

END_FUNCTION_BLOCK

// ---- POUs/Machine/FB_TempLogging_OpcUa.TcPOU
FUNCTION_BLOCK FB_TempLogging_OpcUa
VAR
  // used data
  _pAdsPh  : ARRAY[1..nC_MaxPHs] OF POINTER TO ST_ADS_PH;
  _nRegPhs : UDINT;                                           (*number o registered printheads*)

  // timing
  fb_TonMaxTemp                             : TON;            (*Timer for max temperature*)
  tL_TimeMaxTemp                            : TIME := T#10S;  (*Interval for max temperature*)
  i                                         : UDINT;
  
  {attribute 'OPC.UA.DA':='1'}
  iL_TempActValuePH                         : ARRAY[1..nC_MaxPHs] OF INT;       (*Actual temperature PHx*)
  {attribute 'OPC.UA.DA':='1'}
  iL_TempMaxValuePH                         : ARRAY[1..nC_MaxPHs] OF INT;       (*Max temperature in interval PHx*)
END_VAR
VAR CONSTANT
  nC_MaxPHs                                 : UDINT := 8;
END_VAR

(*Detect max temp value in defined interval*)
fb_TonMaxTemp(IN := NOT fb_TonMaxTemp.Q, PT := tL_TimeMaxTemp);
IF fb_TonMaxTemp.Q THEN
  
  FOR i:=1 TO _nRegPhs DO 
    iL_TempActValuePH[i] := iL_TempMaxValuePH[i];
    iL_TempMaxValuePH[i] := _pAdsPh[i]^.iO_Temperature;
	END_FOR

END_IF

iL_TempMaxValuePH[i] := MAX(iL_TempMaxValuePH[i], _pAdsPh[i]^.iO_Temperature);

METHOD registerPH : BOOL
VAR_INPUT
  pAdsPh : POINTER TO ST_ADS_PH;
END_VAR
IF pAdsPh = 0 THEN RETURN; END_IF 
IF _nRegPhs >= nC_MaxPHs THEN F_LogError('Too many phs already registered'); RETURN; END_IF 


_nRegPhs := _nRegPhs + 1;
_pAdsPh[_nRegPhs] := pAdsPh;
END_METHOD

END_FUNCTION_BLOCK

// ---- POUs/Machine/PowerControl/FB_PowerControl.TcPOU
(*
  PowerSupply control (WAGO Epsitron)
  NOTE: has direct mapped I/Os
*)
FUNCTION_BLOCK FB_PowerControl EXTENDS T_NamedBase
VAR_OUTPUT
  bO_AllFuseOk        : BOOL;
  bO_AllEpsitronOk    : BOOL;
  bO_AllInputOk       : BOOL;
END_VAR
VAR
  i : UDINT;
  
  // Commands
  bAckMsg : BOOL;
  
  // Epsitron Controls
  fbEpsitronFuseControl                     : ARRAY[1..nMaxEpsitrons] OF FB_EpsitronFuseControl;   // internal instances of epsitrons
  // list of epsitron for view & global control
  pEpsitronsInst                            : ARRAY[1..nMaxEpsitrons] OF POINTER TO FB_EpsitronFuseControl;   // list
  bEpsitronsAllChOk                         : ARRAY[1..nMaxEpsitrons] OF BOOL;
  nEpsitronsRegistered                      : UDINT := 0;
  nEpsitronViewSel                          : UDINT := 1;
  
  // Fuse (I/O) supervision
  nFuseInputsRegistered                     : UDINT;
  aFuseNames                                : ARRAY[1..nMaxFuseInputs] OF STRING;
  pFuseInputs                               : ARRAY[1..nMaxFuseInputs] OF POINTER TO BOOL;
  nFuseViewSel                              : UDINT := 1;
END_VAR
VAR CONSTANT
  nMaxEpsitrons : UDINT := 10;
  nMaxFuseInputs : UDINT := 20;
END_VAR

bO_AllEpsitronOk := TRUE;
FOR i:=1 TO nEpsitronsRegistered DO
  IF pEpsitronsInst[i] <> 0 THEN
    pEpsitronsInst[i]^();
    
    bEpsitronsAllChOk[i] := NOT (   (pEpsitronsInst[i]^.iO_Channel1Status = 3)
                              OR (pEpsitronsInst[i]^.iO_Channel2Status = 3)
                              OR (pEpsitronsInst[i]^.iO_Channel3Status = 3)
                              OR (pEpsitronsInst[i]^.iO_Channel4Status = 3));

    
    bO_AllEpsitronOk := bO_AllEpsitronOk AND bEpsitronsAllChOk[i];
  END_IF
END_FOR

// I/O inputs
bO_AllInputOk := TRUE;
FOR i:=1 TO nFuseInputsRegistered DO
  IF pFuseInputs[i] <> 0 THEN
    bO_AllInputOk := bO_AllInputOk AND pFuseInputs[i]^;
  END_IF
END_FOR       

// output
bO_AllFuseOk := bO_AllEpsitronOk AND bO_AllInputOk;
 
// Acknowledge error
IF bAckMsg THEN  bAckMsg := FALSE;
  FOR i:=1 TO nEpsitronsRegistered DO
    pEpsitronsInst[i]^.mAckError();
	END_FOR
END_IF

METHOD ackError
bAckMsg := TRUE;
END_METHOD

(*
  Register configuration for an epsitron directly I/O mapped into this FB.
*)
METHOD registerEpsitron : BOOL
VAR_INPUT
  nInstIdx : UDINT;     // array instance index
  aName    : STRING;    // Epsitron name
  aNameCh1 : STRING;    // name of channel1
  aNameCh2 : STRING;    // name of channel2
  aNameCh3 : STRING;    // name of channel3
  aNameCh4 : STRING;    // name of channel4
END_VAR
IF nInstIdx > nMaxEpsitrons OR nInstIdx = 0      THEN LogError(F_Concat2('registerEpsitron: Invalid index, ignore: ', aName)); END_IF
IF fbEpsitronFuseControl[nInstIdx].aI_Name <> '' THEN LogError(F_Concat2('registerEpsitron: Already configured, ignore: ', aName)); END_IF
IF nEpsitronsRegistered >= nMaxEpsitrons         THEN LogError(F_Concat2('registerEpsitron: Too many already registered, ignore: ', aName)); END_IF
IF aName = ''                                  THEN LogWarning(F_Concat2('registerEpsitron: No name given', '')); END_IF

fbEpsitronFuseControl[nInstIdx].aI_Name := aName;
fbEpsitronFuseControl[nInstIdx].aI_NameChannel1 := aNameCh1;
fbEpsitronFuseControl[nInstIdx].aI_NameChannel2 := aNameCh2;
fbEpsitronFuseControl[nInstIdx].aI_NameChannel3 := aNameCh3;
fbEpsitronFuseControl[nInstIdx].aI_NameChannel4 := aNameCh4;

nEpsitronsRegistered := nEpsitronsRegistered + 1;
pEpsitronsInst[nEpsitronsRegistered] := ADR(fbEpsitronFuseControl[nInstIdx]);

registerEpsitron := TRUE;
END_METHOD

METHOD registerIO : BOOL
VAR_INPUT
  aName  : STRING;              // name of fuse (bool) input
  pInput : POINTER TO BOOL;     // I/O value pointer
END_VAR
IF nFuseInputsRegistered >= nMaxFuseInputs  THEN LogError(F_Concat2('registerIO: Too many already registered, ignore: ', aName)); END_IF
IF pInput = 0                               THEN LogError(F_Concat2('registerIO: Invalid pointer given, ignore: ', aName)); END_IF
IF aName = ''                               THEN LogWarning(F_Concat2('registerIO: No name given', '')); END_IF

nFuseInputsRegistered := nFuseInputsRegistered + 1;
aFuseNames[nFuseInputsRegistered]  := aName;
pFuseInputs[nFuseInputsRegistered] := pInput;

registerIO := TRUE;
END_METHOD

END_FUNCTION_BLOCK

// ---- POUs/Machine/SheetDetectSupervision/FB_SheetDetectSupervision.TcPOU
FUNCTION_BLOCK FB_SheetDetectSupervision
VAR_INPUT
  IbSensorSheetCalender                   AT%I* : BOOL;            // Sensor signal B250
  IbSensorSheetInlet                      AT%I* : BOOL;            // Sensor signal B257
  IbSensorSheetOutlet                     AT%I* : BOOL;            // Sensor signal B254

  InCurrentPos                                  : DINT;            // Current position in [SubPx]
  IbMachineStopped                              : BOOL;            // Machine stopped
  IbInhibitSheetTrigger                         : BOOL;            // inhibit trigger signals for substrate length
  IbCameraTrigger                               : BOOL;            // Camera trigger
  IbMachineSleep                                : BOOL;            // Machine is in Sleep mode
END_VAR

VAR_OUTPUT
  ObSheetJamPrintingSystem                AT%Q* : BOOL;            // Sheet jam in printing system detected

  ObCameraTriggerEnable                         : BOOL;            // Camera trigger enable
  ObCameraTriggerIncorrect                      : BOOL;            // Camera trigger incorrect
  ObCameraTriggerSupervison                     : BOOL;            // Camera trigger supervision for sheet jam
  ObSheetDetectFree                             : BOOL;            // sheet detect sensors are free
END_VAR

VAR
  _PrintSubPixelResolution                      : UDINT := 600 * 32;           // Print sub pixel resolution

  fbSheetDetectRingbuffer01                     : FB_RINGBUFFER;
  fbSheetDetectRingbuffer02                     : FB_RINGBUFFER;

  rfTrig_CameraTriggerSupervison                : RF_TRIG;
  bCameraTriggerSupervisonOn                    : BOOL;
  
  rfTrig_MachineStopped                         : RF_TRIG;

  // jam event
  rTrig_SheetJam                                : R_TRIG;
  _bSheetJamEvent                               : BOOL;

END_VAR

VAR PERSISTENT
  RemSheetDetectSupervisionPar                  : ST_SheetDetectSupervisionPar;
END_VAR

rfTrig_MachineStopped(CLK := IbMachineStopped);

(*B250 => B256*)
fbSheetDetectRingbuffer01.bI_Reset              := IbMachineStopped;
fbSheetDetectRingbuffer01.bI_Sensor             := NOT IbSensorSheetCalender;
fbSheetDetectRingbuffer01.iI_CurrentPos         := DINT_TO_UDINT(InCurrentPos);
fbSheetDetectRingbuffer01.iI_Pg_Offset          := 0;
fbSheetDetectRingbuffer01.iI_Offset_X0          := fbSheetDetectRingbuffer01.iI_CurrentPos + DINT_TO_UDINT(F_MeterToSubPixel(RemSheetDetectSupervisionPar.fR_SheetDetectDistance01, UDINT_TO_LREAL(_PrintSubPixelResolution)));           
fbSheetDetectRingbuffer01.iI_Resolution         := UDINT_TO_INT(_PrintSubPixelResolution);
fbSheetDetectRingbuffer01.fI_ShiftDistance      := 0 - RemSheetDetectSupervisionPar.fR_SheetDetectRange01_m;
fbSheetDetectRingbuffer01();

(*B256 => B254*)
fbSheetDetectRingbuffer02.bI_Reset              := IbMachineStopped;
fbSheetDetectRingbuffer02.bI_Sensor             := IbCameraTrigger;
fbSheetDetectRingbuffer02.iI_CurrentPos         := DINT_TO_UDINT(InCurrentPos);
fbSheetDetectRingbuffer02.iI_Pg_Offset          := 0;
fbSheetDetectRingbuffer02.iI_Offset_X0          := fbSheetDetectRingbuffer02.iI_CurrentPos + DINT_TO_UDINT(F_MeterToSubPixel(RemSheetDetectSupervisionPar.fR_SheetDetectDistance02, UDINT_TO_LREAL(_PrintSubPixelResolution)));           
fbSheetDetectRingbuffer02.iI_Resolution         := UDINT_TO_INT(_PrintSubPixelResolution);
fbSheetDetectRingbuffer02.fI_ShiftDistance      := 0 - RemSheetDetectSupervisionPar.fR_SheetDetectRange02_m;
fbSheetDetectRingbuffer02();

RemSheetDetectSupervisionPar.nR_SheetDetectRange01_SubPx := F_MeterToSubPixel(REAL_TO_LREAL(RemSheetDetectSupervisionPar.fR_SheetDetectRange01_m), UDINT_TO_LREAL(_PrintSubPixelResolution));
RemSheetDetectSupervisionPar.nR_SheetDetectRange02_SubPx := F_MeterToSubPixel(REAL_TO_LREAL(RemSheetDetectSupervisionPar.fR_SheetDetectRange02_m), UDINT_TO_LREAL(_PrintSubPixelResolution));

IF RemSheetDetectSupervisionPar.bR_Enable AND NOT IbMachineSleep THEN
  (*Masking sheet detection of camera system*)
  ObCameraTriggerEnable     :=     (InCurrentPos > (fbSheetDetectRingbuffer01.iO_ShiftOffset_X0 - RemSheetDetectSupervisionPar.nR_SheetDetectRange01_SubPx)) 
                               AND (InCurrentPos < (fbSheetDetectRingbuffer01.iO_ShiftOffset_X0 + RemSheetDetectSupervisionPar.nR_SheetDetectRange01_SubPx));
  (*Sheet trigger was incorrect because of faulty detection*)
  IF NOT ObCameraTriggerEnable AND IbSensorSheetInlet AND NOT IbInhibitSheetTrigger THEN
    ObCameraTriggerIncorrect := TRUE;
  END_IF

  (*Sheet jam supervision*)
  ObCameraTriggerSupervison :=     (InCurrentPos > (fbSheetDetectRingbuffer02.iO_ShiftOffset_X0 - RemSheetDetectSupervisionPar.nR_SheetDetectRange02_SubPx)) 
                               AND (InCurrentPos < (fbSheetDetectRingbuffer02.iO_ShiftOffset_X0 + RemSheetDetectSupervisionPar.nR_SheetDetectRange02_SubPx));
  rfTrig_CameraTriggerSupervison(CLK := ObCameraTriggerSupervison);
  IF rfTrig_CameraTriggerSupervison.RT THEN
    bCameraTriggerSupervisonOn := TRUE;
  END_IF
  IF bCameraTriggerSupervisonOn AND IbSensorSheetOutlet THEN
    bCameraTriggerSupervisonOn := FALSE;
  END_IF
  IF rfTrig_CameraTriggerSupervison.FT AND bCameraTriggerSupervisonOn THEN
    ObSheetJamPrintingSystem   := TRUE;
    bCameraTriggerSupervisonOn := FALSE;
  END_IF

  ObSheetDetectFree := TRUE;
  IF IbMachineStopped THEN
    ObCameraTriggerIncorrect   := FALSE;
    bCameraTriggerSupervisonOn := FALSE;

    IF NOT IbSensorSheetCalender OR IbSensorSheetInlet OR IbSensorSheetOutlet THEN
      ObSheetDetectFree := FALSE;
    END_IF
  END_IF
  IF rfTrig_MachineStopped.RT THEN
    ObSheetJamPrintingSystem   := FALSE;
  END_IF
ELSE
  ObCameraTriggerEnable     := TRUE;
  ObCameraTriggerIncorrect  := FALSE;
  ObSheetJamPrintingSystem  := FALSE;
  ObSheetDetectFree         := TRUE;
END_IF

rTrig_SheetJam(CLK:=ObSheetJamPrintingSystem);
IF rTrig_SheetJam.Q THEN _bSheetJamEvent := TRUE; END_IF

PROPERTY bSheetJamEvent : BOOL
GET
bSheetJamEvent := _bSheetJamEvent;
_bSheetJamEvent := FALSE;
END_GET
END_PROPERTY

PROPERTY PrintSubPixelResolution : UDINT
SET
_PrintSubPixelResolution := PrintSubPixelResolution;
END_SET
END_PROPERTY

END_FUNCTION_BLOCK

